//     PlcTask Inputs/GVL_iXlinker.EtherCAT_Master_EQxxxx.Beckhoff_EQ3xxx.Beckhoff_EQ3xxxEK1122.A_0006_EQ3204_0002_0016.RTD_RTDInputs_Channel_4.Status/Limit_2 <-> RTD RTDInputs Channel 4/Status/Limit 2
//     PlcTask Inputs/GVL_iXlinker.EtherCAT_Master_EQxxxx.Beckhoff_EQ3xxx.Beckhoff_EQ3xxxEK1122.A_0006_EQ3204_0002_0016.RTD_RTDInputs_Channel_1.Status/Error <-> RTD RTDInputs Channel 1/Status/Error
//     PlcTask Inputs/GVL_iXlinker.EtherCAT_Master_EQxxxx.Beckhoff_EQ3xxx.Beckhoff_EQ3xxxEK1122.A_0006_EQ3204_0002_0016.RTD_RTDInputs_Channel_2.Status/Error <-> RTD RTDInputs Channel 2/Status/Error
//     PlcTask Inputs/GVL_iXlinker.EtherCAT_Master_EQxxxx.Beckhoff_EQ3xxx.Beckhoff_EQ3xxxEK1122.A_0006_EQ3204_0002_0016.RTD_RTDInputs_Channel_3.Status/Error <-> RTD RTDInputs Channel 3/Status/Error
//     PlcTask Inputs/GVL_iXlinker.EtherCAT_Master_EQxxxx.Beckhoff_EQ3xxx.Beckhoff_EQ3xxxEK1122.A_0006_EQ3204_0002_0016.RTD_RTDInputs_Channel_4.Status/Error <-> RTD RTDInputs Channel 4/Status/Error
//     PlcTask Inputs/GVL_iXlinker.EtherCAT_Master_EQxxxx.Beckhoff_EQ3xxx.Beckhoff_EQ3xxxEK1122.A_0006_EQ3204_0002_0016.RTD_RTDInputs_Channel_1.Status/Sync_error <-> RTD RTDInputs Channel 1/Status/Sync error
//     PlcTask Inputs/GVL_iXlinker.EtherCAT_Master_EQxxxx.Beckhoff_EQ3xxx.Beckhoff_EQ3xxxEK1122.A_0006_EQ3204_0002_0016.RTD_RTDInputs_Channel_2.Status/Sync_error <-> RTD RTDInputs Channel 2/Status/Sync error
//     PlcTask Inputs/GVL_iXlinker.EtherCAT_Master_EQxxxx.Beckhoff_EQ3xxx.Beckhoff_EQ3xxxEK1122.A_0006_EQ3204_0002_0016.RTD_RTDInputs_Channel_3.Status/Sync_error <-> RTD RTDInputs Channel 3/Status/Sync error
//     PlcTask Inputs/GVL_iXlinker.EtherCAT_Master_EQxxxx.Beckhoff_EQ3xxx.Beckhoff_EQ3xxxEK1122.A_0006_EQ3204_0002_0016.RTD_RTDInputs_Channel_4.Status/Sync_error <-> RTD RTDInputs Channel 4/Status/Sync error
//     PlcTask Inputs/GVL_iXlinker.EtherCAT_Master_EQxxxx.Beckhoff_EQ3xxx.Beckhoff_EQ3xxxEK1122.A_0006_EQ3204_0002_0016.RTD_RTDInputs_Channel_1.Status/TxPDO_State <-> RTD RTDInputs Channel 1/Status/TxPDO State
//     PlcTask Inputs/GVL_iXlinker.EtherCAT_Master_EQxxxx.Beckhoff_EQ3xxx.Beckhoff_EQ3xxxEK1122.A_0006_EQ3204_0002_0016.RTD_RTDInputs_Channel_2.Status/TxPDO_State <-> RTD RTDInputs Channel 2/Status/TxPDO State
//     PlcTask Inputs/GVL_iXlinker.EtherCAT_Master_EQxxxx.Beckhoff_EQ3xxx.Beckhoff_EQ3xxxEK1122.A_0006_EQ3204_0002_0016.RTD_RTDInputs_Channel_3.Status/TxPDO_State <-> RTD RTDInputs Channel 3/Status/TxPDO State
//     PlcTask Inputs/GVL_iXlinker.EtherCAT_Master_EQxxxx.Beckhoff_EQ3xxx.Beckhoff_EQ3xxxEK1122.A_0006_EQ3204_0002_0016.RTD_RTDInputs_Channel_4.Status/TxPDO_State <-> RTD RTDInputs Channel 4/Status/TxPDO State
//     PlcTask Inputs/GVL_iXlinker.EtherCAT_Master_EQxxxx.Beckhoff_EQ3xxx.Beckhoff_EQ3xxxEK1122.A_0006_EQ3204_0002_0016.RTD_RTDInputs_Channel_1.Status/TxPDO_Toggle <-> RTD RTDInputs Channel 1/Status/TxPDO Toggle
//     PlcTask Inputs/GVL_iXlinker.EtherCAT_Master_EQxxxx.Beckhoff_EQ3xxx.Beckhoff_EQ3xxxEK1122.A_0006_EQ3204_0002_0016.RTD_RTDInputs_Channel_2.Status/TxPDO_Toggle <-> RTD RTDInputs Channel 2/Status/TxPDO Toggle
//     PlcTask Inputs/GVL_iXlinker.EtherCAT_Master_EQxxxx.Beckhoff_EQ3xxx.Beckhoff_EQ3xxxEK1122.A_0006_EQ3204_0002_0016.RTD_RTDInputs_Channel_3.Status/TxPDO_Toggle <-> RTD RTDInputs Channel 3/Status/TxPDO Toggle
//     PlcTask Inputs/GVL_iXlinker.EtherCAT_Master_EQxxxx.Beckhoff_EQ3xxx.Beckhoff_EQ3xxxEK1122.A_0006_EQ3204_0002_0016.RTD_RTDInputs_Channel_4.Status/TxPDO_Toggle <-> RTD RTDInputs Channel 4/Status/TxPDO Toggle
//     PlcTask Inputs/GVL_iXlinker.EtherCAT_Master_EQxxxx.Beckhoff_EQ3xxx.Beckhoff_EQ3xxxEK1122.A_0006_EQ3204_0002_0016.RTD_RTDInputs_Channel_1.Value <-> RTD RTDInputs Channel 1/Value
//     PlcTask Inputs/GVL_iXlinker.EtherCAT_Master_EQxxxx.Beckhoff_EQ3xxx.Beckhoff_EQ3xxxEK1122.A_0006_EQ3204_0002_0016.RTD_RTDInputs_Channel_2.Value <-> RTD RTDInputs Channel 2/Value
//     PlcTask Inputs/GVL_iXlinker.EtherCAT_Master_EQxxxx.Beckhoff_EQ3xxx.Beckhoff_EQ3xxxEK1122.A_0006_EQ3204_0002_0016.RTD_RTDInputs_Channel_3.Value <-> RTD RTDInputs Channel 3/Value
//     PlcTask Inputs/GVL_iXlinker.EtherCAT_Master_EQxxxx.Beckhoff_EQ3xxx.Beckhoff_EQ3xxxEK1122.A_0006_EQ3204_0002_0016.RTD_RTDInputs_Channel_4.Value <-> RTD RTDInputs Channel 4/Value
//     PlcTask Inputs/GVL_iXlinker.EtherCAT_Master_EQxxxx.Beckhoff_EQ3xxx.Beckhoff_EQ3xxxEK1122.A_0006_EQ3204_0002_0016.WcState.WcState <-> WcState/WcState
//     PlcTask Inputs/GVL_iXlinker.EtherCAT_Master_EQxxxx.Beckhoff_EQ3xxx.Beckhoff_EQ3xxxEK1122.A_0006_EQ3204_0002_0016.WcState.InputToggle <-> WcState/InputToggle
//     PlcTask Inputs/GVL_iXlinker.EtherCAT_Master_EQxxxx.Beckhoff_EQ3xxx.Beckhoff_EQ3xxxEK1122.A_0006_EQ3204_0002_0016.InfoData.AdsAddr <-> InfoData/AdsAddr
//     PlcTask Inputs/GVL_iXlinker.EtherCAT_Master_EQxxxx.Beckhoff_EQ3xxx.Beckhoff_EQ3xxxEK1122.A_0006_EQ3204_0002_0016.InfoData.State <-> InfoData/State
//   PLC/PLC Instance <-> EtherCAT Master EQxxxx/Beckhoff EQ3xxx/Beckhoff EQ3xxxEK1122/A_0007(EQ3204-0002-0017)
//     PlcTask Inputs/GVL_iXlinker.EtherCAT_Master_EQxxxx.Beckhoff_EQ3xxx.Beckhoff_EQ3xxxEK1122.A_0007_EQ3204_0002_0017.RTD_RTDInputs_Channel_1.Status/Underrange <-> RTD RTDInputs Channel 1/Status/Underrange
//     PlcTask Inputs/GVL_iXlinker.EtherCAT_Master_EQxxxx.Beckhoff_EQ3xxx.Beckhoff_EQ3xxxEK1122.A_0007_EQ3204_0002_0017.RTD_RTDInputs_Channel_2.Status/Underrange <-> RTD RTDInputs Channel 2/Status/Underrange
//     PlcTask Inputs/GVL_iXlinker.EtherCAT_Master_EQxxxx.Beckhoff_EQ3xxx.Beckhoff_EQ3xxxEK1122.A_0007_EQ3204_0002_0017.RTD_RTDInputs_Channel_3.Status/Underrange <-> RTD RTDInputs Channel 3/Status/Underrange
//     PlcTask Inputs/GVL_iXlinker.EtherCAT_Master_EQxxxx.Beckhoff_EQ3xxx.Beckhoff_EQ3xxxEK1122.A_0007_EQ3204_0002_0017.RTD_RTDInputs_Channel_4.Status/Underrange <-> RTD RTDInputs Channel 4/Status/Underrange
//     PlcTask Inputs/GVL_iXlinker.EtherCAT_Master_EQxxxx.Beckhoff_EQ3xxx.Beckhoff_EQ3xxxEK1122.A_0007_EQ3204_0002_0017.RTD_RTDInputs_Channel_1.Status/Overrange <-> RTD RTDInputs Channel 1/Status/Overrange
//     PlcTask Inputs/GVL_iXlinker.EtherCAT_Master_EQxxxx.Beckhoff_EQ3xxx.Beckhoff_EQ3xxxEK1122.A_0007_EQ3204_0002_0017.RTD_RTDInputs_Channel_2.Status/Overrange <-> RTD RTDInputs Channel 2/Status/Overrange
//     PlcTask Inputs/GVL_iXlinker.EtherCAT_Master_EQxxxx.Beckhoff_EQ3xxx.Beckhoff_EQ3xxxEK1122.A_0007_EQ3204_0002_0017.RTD_RTDInputs_Channel_3.Status/Overrange <-> RTD RTDInputs Channel 3/Status/Overrange
//     PlcTask Inputs/GVL_iXlinker.EtherCAT_Master_EQxxxx.Beckhoff_EQ3xxx.Beckhoff_EQ3xxxEK1122.A_0007_EQ3204_0002_0017.RTD_RTDInputs_Channel_4.Status/Overrange <-> RTD RTDInputs Channel 4/Status/Overrange
//     PlcTask Inputs/GVL_iXlinker.EtherCAT_Master_EQxxxx.Beckhoff_EQ3xxx.Beckhoff_EQ3xxxEK1122.A_0007_EQ3204_0002_0017.RTD_RTDInputs_Channel_1.Status/Limit_1 <-> RTD RTDInputs Channel 1/Status/Limit 1
//     PlcTask Inputs/GVL_iXlinker.EtherCAT_Master_EQxxxx.Beckhoff_EQ3xxx.Beckhoff_EQ3xxxEK1122.A_0007_EQ3204_0002_0017.RTD_RTDInputs_Channel_1.Status/Limit_2 <-> RTD RTDInputs Channel 1/Status/Limit 2
//     PlcTask Inputs/GVL_iXlinker.EtherCAT_Master_EQxxxx.Beckhoff_EQ3xxx.Beckhoff_EQ3xxxEK1122.A_0007_EQ3204_0002_0017.RTD_RTDInputs_Channel_2.Status/Limit_1 <-> RTD RTDInputs Channel 2/Status/Limit 1
//     PlcTask Inputs/GVL_iXlinker.EtherCAT_Master_EQxxxx.Beckhoff_EQ3xxx.Beckhoff_EQ3xxxEK1122.A_0007_EQ3204_0002_0017.RTD_RTDInputs_Channel_2.Status/Limit_2 <-> RTD RTDInputs Channel 2/Status/Limit 2
//     PlcTask Inputs/GVL_iXlinker.EtherCAT_Master_EQxxxx.Beckhoff_EQ3xxx.Beckhoff_EQ3xxxEK1122.A_0007_EQ3204_0002_0017.RTD_RTDInputs_Channel_3.Status/Limit_1 <-> RTD RTDInputs Channel 3/Status/Limit 1
//     PlcTask Inputs/GVL_iXlinker.EtherCAT_Master_EQxxxx.Beckhoff_EQ3xxx.Beckhoff_EQ3xxxEK1122.A_0007_EQ3204_0002_0017.RTD_RTDInputs_Channel_3.Status/Limit_2 <-> RTD RTDInputs Channel 3/Status/Limit 2
//     PlcTask Inputs/GVL_iXlinker.EtherCAT_Master_EQxxxx.Beckhoff_EQ3xxx.Beckhoff_EQ3xxxEK1122.A_0007_EQ3204_0002_0017.RTD_RTDInputs_Channel_4.Status/Limit_1 <-> RTD RTDInputs Channel 4/Status/Limit 1
//     PlcTask Inputs/GVL_iXlinker.EtherCAT_Master_EQxxxx.Beckhoff_EQ3xxx.Beckhoff_EQ3xxxEK1122.A_0007_EQ3204_0002_0017.RTD_RTDInputs_Channel_4.Status/Limit_2 <-> RTD RTDInputs Channel 4/Status/Limit 2
//     PlcTask Inputs/GVL_iXlinker.EtherCAT_Master_EQxxxx.Beckhoff_EQ3xxx.Beckhoff_EQ3xxxEK1122.A_0007_EQ3204_0002_0017.RTD_RTDInputs_Channel_1.Status/Error <-> RTD RTDInputs Channel 1/Status/Error
//     PlcTask Inputs/GVL_iXlinker.EtherCAT_Master_EQxxxx.Beckhoff_EQ3xxx.Beckhoff_EQ3xxxEK1122.A_0007_EQ3204_0002_0017.RTD_RTDInputs_Channel_2.Status/Error <-> RTD RTDInputs Channel 2/Status/Error
//     PlcTask Inputs/GVL_iXlinker.EtherCAT_Master_EQxxxx.Beckhoff_EQ3xxx.Beckhoff_EQ3xxxEK1122.A_0007_EQ3204_0002_0017.RTD_RTDInputs_Channel_3.Status/Error <-> RTD RTDInputs Channel 3/Status/Error
//     PlcTask Inputs/GVL_iXlinker.EtherCAT_Master_EQxxxx.Beckhoff_EQ3xxx.Beckhoff_EQ3xxxEK1122.A_0007_EQ3204_0002_0017.RTD_RTDInputs_Channel_4.Status/Error <-> RTD RTDInputs Channel 4/Status/Error
//     PlcTask Inputs/GVL_iXlinker.EtherCAT_Master_EQxxxx.Beckhoff_EQ3xxx.Beckhoff_EQ3xxxEK1122.A_0007_EQ3204_0002_0017.RTD_RTDInputs_Channel_1.Status/Sync_error <-> RTD RTDInputs Channel 1/Status/Sync error
//     PlcTask Inputs/GVL_iXlinker.EtherCAT_Master_EQxxxx.Beckhoff_EQ3xxx.Beckhoff_EQ3xxxEK1122.A_0007_EQ3204_0002_0017.RTD_RTDInputs_Channel_2.Status/Sync_error <-> RTD RTDInputs Channel 2/Status/Sync error
//     PlcTask Inputs/GVL_iXlinker.EtherCAT_Master_EQxxxx.Beckhoff_EQ3xxx.Beckhoff_EQ3xxxEK1122.A_0007_EQ3204_0002_0017.RTD_RTDInputs_Channel_3.Status/Sync_error <-> RTD RTDInputs Channel 3/Status/Sync error
//     PlcTask Inputs/GVL_iXlinker.EtherCAT_Master_EQxxxx.Beckhoff_EQ3xxx.Beckhoff_EQ3xxxEK1122.A_0007_EQ3204_0002_0017.RTD_RTDInputs_Channel_4.Status/Sync_error <-> RTD RTDInputs Channel 4/Status/Sync error
//     PlcTask Inputs/GVL_iXlinker.EtherCAT_Master_EQxxxx.Beckhoff_EQ3xxx.Beckhoff_EQ3xxxEK1122.A_0007_EQ3204_0002_0017.RTD_RTDInputs_Channel_1.Status/TxPDO_State <-> RTD RTDInputs Channel 1/Status/TxPDO State
//     PlcTask Inputs/GVL_iXlinker.EtherCAT_Master_EQxxxx.Beckhoff_EQ3xxx.Beckhoff_EQ3xxxEK1122.A_0007_EQ3204_0002_0017.RTD_RTDInputs_Channel_2.Status/TxPDO_State <-> RTD RTDInputs Channel 2/Status/TxPDO State
//     PlcTask Inputs/GVL_iXlinker.EtherCAT_Master_EQxxxx.Beckhoff_EQ3xxx.Beckhoff_EQ3xxxEK1122.A_0007_EQ3204_0002_0017.RTD_RTDInputs_Channel_3.Status/TxPDO_State <-> RTD RTDInputs Channel 3/Status/TxPDO State
//     PlcTask Inputs/GVL_iXlinker.EtherCAT_Master_EQxxxx.Beckhoff_EQ3xxx.Beckhoff_EQ3xxxEK1122.A_0007_EQ3204_0002_0017.RTD_RTDInputs_Channel_4.Status/TxPDO_State <-> RTD RTDInputs Channel 4/Status/TxPDO State
//     PlcTask Inputs/GVL_iXlinker.EtherCAT_Master_EQxxxx.Beckhoff_EQ3xxx.Beckhoff_EQ3xxxEK1122.A_0007_EQ3204_0002_0017.RTD_RTDInputs_Channel_1.Status/TxPDO_Toggle <-> RTD RTDInputs Channel 1/Status/TxPDO Toggle
//     PlcTask Inputs/GVL_iXlinker.EtherCAT_Master_EQxxxx.Beckhoff_EQ3xxx.Beckhoff_EQ3xxxEK1122.A_0007_EQ3204_0002_0017.RTD_RTDInputs_Channel_2.Status/TxPDO_Toggle <-> RTD RTDInputs Channel 2/Status/TxPDO Toggle
//     PlcTask Inputs/GVL_iXlinker.EtherCAT_Master_EQxxxx.Beckhoff_EQ3xxx.Beckhoff_EQ3xxxEK1122.A_0007_EQ3204_0002_0017.RTD_RTDInputs_Channel_3.Status/TxPDO_Toggle <-> RTD RTDInputs Channel 3/Status/TxPDO Toggle
//     PlcTask Inputs/GVL_iXlinker.EtherCAT_Master_EQxxxx.Beckhoff_EQ3xxx.Beckhoff_EQ3xxxEK1122.A_0007_EQ3204_0002_0017.RTD_RTDInputs_Channel_4.Status/TxPDO_Toggle <-> RTD RTDInputs Channel 4/Status/TxPDO Toggle
//     PlcTask Inputs/GVL_iXlinker.EtherCAT_Master_EQxxxx.Beckhoff_EQ3xxx.Beckhoff_EQ3xxxEK1122.A_0007_EQ3204_0002_0017.RTD_RTDInputs_Channel_1.Value <-> RTD RTDInputs Channel 1/Value
//     PlcTask Inputs/GVL_iXlinker.EtherCAT_Master_EQxxxx.Beckhoff_EQ3xxx.Beckhoff_EQ3xxxEK1122.A_0007_EQ3204_0002_0017.RTD_RTDInputs_Channel_2.Value <-> RTD RTDInputs Channel 2/Value
//     PlcTask Inputs/GVL_iXlinker.EtherCAT_Master_EQxxxx.Beckhoff_EQ3xxx.Beckhoff_EQ3xxxEK1122.A_0007_EQ3204_0002_0017.RTD_RTDInputs_Channel_3.Value <-> RTD RTDInputs Channel 3/Value
//     PlcTask Inputs/GVL_iXlinker.EtherCAT_Master_EQxxxx.Beckhoff_EQ3xxx.Beckhoff_EQ3xxxEK1122.A_0007_EQ3204_0002_0017.RTD_RTDInputs_Channel_4.Value <-> RTD RTDInputs Channel 4/Value
//     PlcTask Inputs/GVL_iXlinker.EtherCAT_Master_EQxxxx.Beckhoff_EQ3xxx.Beckhoff_EQ3xxxEK1122.A_0007_EQ3204_0002_0017.WcState.WcState <-> WcState/WcState
//     PlcTask Inputs/GVL_iXlinker.EtherCAT_Master_EQxxxx.Beckhoff_EQ3xxx.Beckhoff_EQ3xxxEK1122.A_0007_EQ3204_0002_0017.WcState.InputToggle <-> WcState/InputToggle
//     PlcTask Inputs/GVL_iXlinker.EtherCAT_Master_EQxxxx.Beckhoff_EQ3xxx.Beckhoff_EQ3xxxEK1122.A_0007_EQ3204_0002_0017.InfoData.AdsAddr <-> InfoData/AdsAddr
//     PlcTask Inputs/GVL_iXlinker.EtherCAT_Master_EQxxxx.Beckhoff_EQ3xxx.Beckhoff_EQ3xxxEK1122.A_0007_EQ3204_0002_0017.InfoData.State <-> InfoData/State
//   PLC/PLC Instance <-> EtherCAT Master EQxxxx/Beckhoff EQ3xxx/Beckhoff EQ3xxxEK1122/A_0008(EQ3204-0002-0020)
//     PlcTask Inputs/GVL_iXlinker.EtherCAT_Master_EQxxxx.Beckhoff_EQ3xxx.Beckhoff_EQ3xxxEK1122.A_0008_EQ3204_0002_0020.RTD_RTDInputs_Channel_1.Status/Underrange <-> RTD RTDInputs Channel 1/Status/Underrange
//     PlcTask Inputs/GVL_iXlinker.EtherCAT_Master_EQxxxx.Beckhoff_EQ3xxx.Beckhoff_EQ3xxxEK1122.A_0008_EQ3204_0002_0020.RTD_RTDInputs_Channel_2.Status/Underrange <-> RTD RTDInputs Channel 2/Status/Underrange
//     PlcTask Inputs/GVL_iXlinker.EtherCAT_Master_EQxxxx.Beckhoff_EQ3xxx.Beckhoff_EQ3xxxEK1122.A_0008_EQ3204_0002_0020.RTD_RTDInputs_Channel_3.Status/Underrange <-> RTD RTDInputs Channel 3/Status/Underrange
//     PlcTask Inputs/GVL_iXlinker.EtherCAT_Master_EQxxxx.Beckhoff_EQ3xxx.Beckhoff_EQ3xxxEK1122.A_0008_EQ3204_0002_0020.RTD_RTDInputs_Channel_4.Status/Underrange <-> RTD RTDInputs Channel 4/Status/Underrange
//     PlcTask Inputs/GVL_iXlinker.EtherCAT_Master_EQxxxx.Beckhoff_EQ3xxx.Beckhoff_EQ3xxxEK1122.A_0008_EQ3204_0002_0020.RTD_RTDInputs_Channel_1.Status/Overrange <-> RTD RTDInputs Channel 1/Status/Overrange
//     PlcTask Inputs/GVL_iXlinker.EtherCAT_Master_EQxxxx.Beckhoff_EQ3xxx.Beckhoff_EQ3xxxEK1122.A_0008_EQ3204_0002_0020.RTD_RTDInputs_Channel_2.Status/Overrange <-> RTD RTDInputs Channel 2/Status/Overrange
//     PlcTask Inputs/GVL_iXlinker.EtherCAT_Master_EQxxxx.Beckhoff_EQ3xxx.Beckhoff_EQ3xxxEK1122.A_0008_EQ3204_0002_0020.RTD_RTDInputs_Channel_3.Status/Overrange <-> RTD RTDInputs Channel 3/Status/Overrange
//     PlcTask Inputs/GVL_iXlinker.EtherCAT_Master_EQxxxx.Beckhoff_EQ3xxx.Beckhoff_EQ3xxxEK1122.A_0008_EQ3204_0002_0020.RTD_RTDInputs_Channel_4.Status/Overrange <-> RTD RTDInputs Channel 4/Status/Overrange
//     PlcTask Inputs/GVL_iXlinker.EtherCAT_Master_EQxxxx.Beckhoff_EQ3xxx.Beckhoff_EQ3xxxEK1122.A_0008_EQ3204_0002_0020.RTD_RTDInputs_Channel_1.Status/Limit_1 <-> RTD RTDInputs Channel 1/Status/Limit 1
//     PlcTask Inputs/GVL_iXlinker.EtherCAT_Master_EQxxxx.Beckhoff_EQ3xxx.Beckhoff_EQ3xxxEK1122.A_0008_EQ3204_0002_0020.RTD_RTDInputs_Channel_1.Status/Limit_2 <-> RTD RTDInputs Channel 1/Status/Limit 2
//     PlcTask Inputs/GVL_iXlinker.EtherCAT_Master_EQxxxx.Beckhoff_EQ3xxx.Beckhoff_EQ3xxxEK1122.A_0008_EQ3204_0002_0020.RTD_RTDInputs_Channel_2.Status/Limit_1 <-> RTD RTDInputs Channel 2/Status/Limit 1
//     PlcTask Inputs/GVL_iXlinker.EtherCAT_Master_EQxxxx.Beckhoff_EQ3xxx.Beckhoff_EQ3xxxEK1122.A_0008_EQ3204_0002_0020.RTD_RTDInputs_Channel_2.Status/Limit_2 <-> RTD RTDInputs Channel 2/Status/Limit 2
//     PlcTask Inputs/GVL_iXlinker.EtherCAT_Master_EQxxxx.Beckhoff_EQ3xxx.Beckhoff_EQ3xxxEK1122.A_0008_EQ3204_0002_0020.RTD_RTDInputs_Channel_3.Status/Limit_1 <-> RTD RTDInputs Channel 3/Status/Limit 1
//     PlcTask Inputs/GVL_iXlinker.EtherCAT_Master_EQxxxx.Beckhoff_EQ3xxx.Beckhoff_EQ3xxxEK1122.A_0008_EQ3204_0002_0020.RTD_RTDInputs_Channel_3.Status/Limit_2 <-> RTD RTDInputs Channel 3/Status/Limit 2
//     PlcTask Inputs/GVL_iXlinker.EtherCAT_Master_EQxxxx.Beckhoff_EQ3xxx.Beckhoff_EQ3xxxEK1122.A_0008_EQ3204_0002_0020.RTD_RTDInputs_Channel_4.Status/Limit_1 <-> RTD RTDInputs Channel 4/Status/Limit 1
//     PlcTask Inputs/GVL_iXlinker.EtherCAT_Master_EQxxxx.Beckhoff_EQ3xxx.Beckhoff_EQ3xxxEK1122.A_0008_EQ3204_0002_0020.RTD_RTDInputs_Channel_4.Status/Limit_2 <-> RTD RTDInputs Channel 4/Status/Limit 2
//     PlcTask Inputs/GVL_iXlinker.EtherCAT_Master_EQxxxx.Beckhoff_EQ3xxx.Beckhoff_EQ3xxxEK1122.A_0008_EQ3204_0002_0020.RTD_RTDInputs_Channel_1.Status/Error <-> RTD RTDInputs Channel 1/Status/Error
//     PlcTask Inputs/GVL_iXlinker.EtherCAT_Master_EQxxxx.Beckhoff_EQ3xxx.Beckhoff_EQ3xxxEK1122.A_0008_EQ3204_0002_0020.RTD_RTDInputs_Channel_2.Status/Error <-> RTD RTDInputs Channel 2/Status/Error
//     PlcTask Inputs/GVL_iXlinker.EtherCAT_Master_EQxxxx.Beckhoff_EQ3xxx.Beckhoff_EQ3xxxEK1122.A_0008_EQ3204_0002_0020.RTD_RTDInputs_Channel_3.Status/Error <-> RTD RTDInputs Channel 3/Status/Error
//     PlcTask Inputs/GVL_iXlinker.EtherCAT_Master_EQxxxx.Beckhoff_EQ3xxx.Beckhoff_EQ3xxxEK1122.A_0008_EQ3204_0002_0020.RTD_RTDInputs_Channel_4.Status/Error <-> RTD RTDInputs Channel 4/Status/Error
//     PlcTask Inputs/GVL_iXlinker.EtherCAT_Master_EQxxxx.Beckhoff_EQ3xxx.Beckhoff_EQ3xxxEK1122.A_0008_EQ3204_0002_0020.RTD_RTDInputs_Channel_1.Status/Sync_error <-> RTD RTDInputs Channel 1/Status/Sync error
//     PlcTask Inputs/GVL_iXlinker.EtherCAT_Master_EQxxxx.Beckhoff_EQ3xxx.Beckhoff_EQ3xxxEK1122.A_0008_EQ3204_0002_0020.RTD_RTDInputs_Channel_2.Status/Sync_error <-> RTD RTDInputs Channel 2/Status/Sync error
//     PlcTask Inputs/GVL_iXlinker.EtherCAT_Master_EQxxxx.Beckhoff_EQ3xxx.Beckhoff_EQ3xxxEK1122.A_0008_EQ3204_0002_0020.RTD_RTDInputs_Channel_3.Status/Sync_error <-> RTD RTDInputs Channel 3/Status/Sync error
//     PlcTask Inputs/GVL_iXlinker.EtherCAT_Master_EQxxxx.Beckhoff_EQ3xxx.Beckhoff_EQ3xxxEK1122.A_0008_EQ3204_0002_0020.RTD_RTDInputs_Channel_4.Status/Sync_error <-> RTD RTDInputs Channel 4/Status/Sync error
//     PlcTask Inputs/GVL_iXlinker.EtherCAT_Master_EQxxxx.Beckhoff_EQ3xxx.Beckhoff_EQ3xxxEK1122.A_0008_EQ3204_0002_0020.RTD_RTDInputs_Channel_1.Status/TxPDO_State <-> RTD RTDInputs Channel 1/Status/TxPDO State
//     PlcTask Inputs/GVL_iXlinker.EtherCAT_Master_EQxxxx.Beckhoff_EQ3xxx.Beckhoff_EQ3xxxEK1122.A_0008_EQ3204_0002_0020.RTD_RTDInputs_Channel_2.Status/TxPDO_State <-> RTD RTDInputs Channel 2/Status/TxPDO State
//     PlcTask Inputs/GVL_iXlinker.EtherCAT_Master_EQxxxx.Beckhoff_EQ3xxx.Beckhoff_EQ3xxxEK1122.A_0008_EQ3204_0002_0020.RTD_RTDInputs_Channel_3.Status/TxPDO_State <-> RTD RTDInputs Channel 3/Status/TxPDO State
//     PlcTask Inputs/GVL_iXlinker.EtherCAT_Master_EQxxxx.Beckhoff_EQ3xxx.Beckhoff_EQ3xxxEK1122.A_0008_EQ3204_0002_0020.RTD_RTDInputs_Channel_4.Status/TxPDO_State <-> RTD RTDInputs Channel 4/Status/TxPDO State
//     PlcTask Inputs/GVL_iXlinker.EtherCAT_Master_EQxxxx.Beckhoff_EQ3xxx.Beckhoff_EQ3xxxEK1122.A_0008_EQ3204_0002_0020.RTD_RTDInputs_Channel_1.Status/TxPDO_Toggle <-> RTD RTDInputs Channel 1/Status/TxPDO Toggle
//     PlcTask Inputs/GVL_iXlinker.EtherCAT_Master_EQxxxx.Beckhoff_EQ3xxx.Beckhoff_EQ3xxxEK1122.A_0008_EQ3204_0002_0020.RTD_RTDInputs_Channel_2.Status/TxPDO_Toggle <-> RTD RTDInputs Channel 2/Status/TxPDO Toggle
//     PlcTask Inputs/GVL_iXlinker.EtherCAT_Master_EQxxxx.Beckhoff_EQ3xxx.Beckhoff_EQ3xxxEK1122.A_0008_EQ3204_0002_0020.RTD_RTDInputs_Channel_3.Status/TxPDO_Toggle <-> RTD RTDInputs Channel 3/Status/TxPDO Toggle
//     PlcTask Inputs/GVL_iXlinker.EtherCAT_Master_EQxxxx.Beckhoff_EQ3xxx.Beckhoff_EQ3xxxEK1122.A_0008_EQ3204_0002_0020.RTD_RTDInputs_Channel_4.Status/TxPDO_Toggle <-> RTD RTDInputs Channel 4/Status/TxPDO Toggle
//     PlcTask Inputs/GVL_iXlinker.EtherCAT_Master_EQxxxx.Beckhoff_EQ3xxx.Beckhoff_EQ3xxxEK1122.A_0008_EQ3204_0002_0020.RTD_RTDInputs_Channel_1.Value <-> RTD RTDInputs Channel 1/Value
//     PlcTask Inputs/GVL_iXlinker.EtherCAT_Master_EQxxxx.Beckhoff_EQ3xxx.Beckhoff_EQ3xxxEK1122.A_0008_EQ3204_0002_0020.RTD_RTDInputs_Channel_2.Value <-> RTD RTDInputs Channel 2/Value
//     PlcTask Inputs/GVL_iXlinker.EtherCAT_Master_EQxxxx.Beckhoff_EQ3xxx.Beckhoff_EQ3xxxEK1122.A_0008_EQ3204_0002_0020.RTD_RTDInputs_Channel_3.Value <-> RTD RTDInputs Channel 3/Value
//     PlcTask Inputs/GVL_iXlinker.EtherCAT_Master_EQxxxx.Beckhoff_EQ3xxx.Beckhoff_EQ3xxxEK1122.A_0008_EQ3204_0002_0020.RTD_RTDInputs_Channel_4.Value <-> RTD RTDInputs Channel 4/Value
//     PlcTask Inputs/GVL_iXlinker.EtherCAT_Master_EQxxxx.Beckhoff_EQ3xxx.Beckhoff_EQ3xxxEK1122.A_0008_EQ3204_0002_0020.WcState.WcState <-> WcState/WcState
//     PlcTask Inputs/GVL_iXlinker.EtherCAT_Master_EQxxxx.Beckhoff_EQ3xxx.Beckhoff_EQ3xxxEK1122.A_0008_EQ3204_0002_0020.WcState.InputToggle <-> WcState/InputToggle
//     PlcTask Inputs/GVL_iXlinker.EtherCAT_Master_EQxxxx.Beckhoff_EQ3xxx.Beckhoff_EQ3xxxEK1122.A_0008_EQ3204_0002_0020.InfoData.AdsAddr <-> InfoData/AdsAddr
//     PlcTask Inputs/GVL_iXlinker.EtherCAT_Master_EQxxxx.Beckhoff_EQ3xxx.Beckhoff_EQ3xxxEK1122.A_0008_EQ3204_0002_0020.InfoData.State <-> InfoData/State
//   PLC/PLC Instance <-> EtherCAT Master EQxxxx/Beckhoff EQ3xxx/Beckhoff EQ3xxxEK1122/A_0009(EQ3204-0002-0021)
//     PlcTask Inputs/GVL_iXlinker.EtherCAT_Master_EQxxxx.Beckhoff_EQ3xxx.Beckhoff_EQ3xxxEK1122.A_0009_EQ3204_0002_0021.RTD_RTDInputs_Channel_1.Status/Underrange <-> RTD RTDInputs Channel 1/Status/Underrange
//     PlcTask Inputs/GVL_iXlinker.EtherCAT_Master_EQxxxx.Beckhoff_EQ3xxx.Beckhoff_EQ3xxxEK1122.A_0009_EQ3204_0002_0021.RTD_RTDInputs_Channel_2.Status/Underrange <-> RTD RTDInputs Channel 2/Status/Underrange
//     PlcTask Inputs/GVL_iXlinker.EtherCAT_Master_EQxxxx.Beckhoff_EQ3xxx.Beckhoff_EQ3xxxEK1122.A_0009_EQ3204_0002_0021.RTD_RTDInputs_Channel_3.Status/Underrange <-> RTD RTDInputs Channel 3/Status/Underrange
//     PlcTask Inputs/GVL_iXlinker.EtherCAT_Master_EQxxxx.Beckhoff_EQ3xxx.Beckhoff_EQ3xxxEK1122.A_0009_EQ3204_0002_0021.RTD_RTDInputs_Channel_4.Status/Underrange <-> RTD RTDInputs Channel 4/Status/Underrange
//     PlcTask Inputs/GVL_iXlinker.EtherCAT_Master_EQxxxx.Beckhoff_EQ3xxx.Beckhoff_EQ3xxxEK1122.A_0009_EQ3204_0002_0021.RTD_RTDInputs_Channel_1.Status/Overrange <-> RTD RTDInputs Channel 1/Status/Overrange
//     PlcTask Inputs/GVL_iXlinker.EtherCAT_Master_EQxxxx.Beckhoff_EQ3xxx.Beckhoff_EQ3xxxEK1122.A_0009_EQ3204_0002_0021.RTD_RTDInputs_Channel_2.Status/Overrange <-> RTD RTDInputs Channel 2/Status/Overrange
//     PlcTask Inputs/GVL_iXlinker.EtherCAT_Master_EQxxxx.Beckhoff_EQ3xxx.Beckhoff_EQ3xxxEK1122.A_0009_EQ3204_0002_0021.RTD_RTDInputs_Channel_3.Status/Overrange <-> RTD RTDInputs Channel 3/Status/Overrange
//     PlcTask Inputs/GVL_iXlinker.EtherCAT_Master_EQxxxx.Beckhoff_EQ3xxx.Beckhoff_EQ3xxxEK1122.A_0009_EQ3204_0002_0021.RTD_RTDInputs_Channel_4.Status/Overrange <-> RTD RTDInputs Channel 4/Status/Overrange
//     PlcTask Inputs/GVL_iXlinker.EtherCAT_Master_EQxxxx.Beckhoff_EQ3xxx.Beckhoff_EQ3xxxEK1122.A_0009_EQ3204_0002_0021.RTD_RTDInputs_Channel_1.Status/Limit_1 <-> RTD RTDInputs Channel 1/Status/Limit 1
//     PlcTask Inputs/GVL_iXlinker.EtherCAT_Master_EQxxxx.Beckhoff_EQ3xxx.Beckhoff_EQ3xxxEK1122.A_0009_EQ3204_0002_0021.RTD_RTDInputs_Channel_1.Status/Limit_2 <-> RTD RTDInputs Channel 1/Status/Limit 2
//     PlcTask Inputs/GVL_iXlinker.EtherCAT_Master_EQxxxx.Beckhoff_EQ3xxx.Beckhoff_EQ3xxxEK1122.A_0009_EQ3204_0002_0021.RTD_RTDInputs_Channel_2.Status/Limit_1 <-> RTD RTDInputs Channel 2/Status/Limit 1
//     PlcTask Inputs/GVL_iXlinker.EtherCAT_Master_EQxxxx.Beckhoff_EQ3xxx.Beckhoff_EQ3xxxEK1122.A_0009_EQ3204_0002_0021.RTD_RTDInputs_Channel_2.Status/Limit_2 <-> RTD RTDInputs Channel 2/Status/Limit 2
//     PlcTask Inputs/GVL_iXlinker.EtherCAT_Master_EQxxxx.Beckhoff_EQ3xxx.Beckhoff_EQ3xxxEK1122.A_0009_EQ3204_0002_0021.RTD_RTDInputs_Channel_3.Status/Limit_1 <-> RTD RTDInputs Channel 3/Status/Limit 1
//     PlcTask Inputs/GVL_iXlinker.EtherCAT_Master_EQxxxx.Beckhoff_EQ3xxx.Beckhoff_EQ3xxxEK1122.A_0009_EQ3204_0002_0021.RTD_RTDInputs_Channel_3.Status/Limit_2 <-> RTD RTDInputs Channel 3/Status/Limit 2
//     PlcTask Inputs/GVL_iXlinker.EtherCAT_Master_EQxxxx.Beckhoff_EQ3xxx.Beckhoff_EQ3xxxEK1122.A_0009_EQ3204_0002_0021.RTD_RTDInputs_Channel_4.Status/Limit_1 <-> RTD RTDInputs Channel 4/Status/Limit 1
//     PlcTask Inputs/GVL_iXlinker.EtherCAT_Master_EQxxxx.Beckhoff_EQ3xxx.Beckhoff_EQ3xxxEK1122.A_0009_EQ3204_0002_0021.RTD_RTDInputs_Channel_4.Status/Limit_2 <-> RTD RTDInputs Channel 4/Status/Limit 2
//     PlcTask Inputs/GVL_iXlinker.EtherCAT_Master_EQxxxx.Beckhoff_EQ3xxx.Beckhoff_EQ3xxxEK1122.A_0009_EQ3204_0002_0021.RTD_RTDInputs_Channel_1.Status/Error <-> RTD RTDInputs Channel 1/Status/Error
//     PlcTask Inputs/GVL_iXlinker.EtherCAT_Master_EQxxxx.Beckhoff_EQ3xxx.Beckhoff_EQ3xxxEK1122.A_0009_EQ3204_0002_0021.RTD_RTDInputs_Channel_2.Status/Error <-> RTD RTDInputs Channel 2/Status/Error
//     PlcTask Inputs/GVL_iXlinker.EtherCAT_Master_EQxxxx.Beckhoff_EQ3xxx.Beckhoff_EQ3xxxEK1122.A_0009_EQ3204_0002_0021.RTD_RTDInputs_Channel_3.Status/Error <-> RTD RTDInputs Channel 3/Status/Error
//     PlcTask Inputs/GVL_iXlinker.EtherCAT_Master_EQxxxx.Beckhoff_EQ3xxx.Beckhoff_EQ3xxxEK1122.A_0009_EQ3204_0002_0021.RTD_RTDInputs_Channel_4.Status/Error <-> RTD RTDInputs Channel 4/Status/Error
//     PlcTask Inputs/GVL_iXlinker.EtherCAT_Master_EQxxxx.Beckhoff_EQ3xxx.Beckhoff_EQ3xxxEK1122.A_0009_EQ3204_0002_0021.RTD_RTDInputs_Channel_1.Status/TxPDO_State <-> RTD RTDInputs Channel 1/Status/TxPDO State
//     PlcTask Inputs/GVL_iXlinker.EtherCAT_Master_EQxxxx.Beckhoff_EQ3xxx.Beckhoff_EQ3xxxEK1122.A_0009_EQ3204_0002_0021.RTD_RTDInputs_Channel_2.Status/TxPDO_State <-> RTD RTDInputs Channel 2/Status/TxPDO State
//     PlcTask Inputs/GVL_iXlinker.EtherCAT_Master_EQxxxx.Beckhoff_EQ3xxx.Beckhoff_EQ3xxxEK1122.A_0009_EQ3204_0002_0021.RTD_RTDInputs_Channel_3.Status/TxPDO_State <-> RTD RTDInputs Channel 3/Status/TxPDO State
//     PlcTask Inputs/GVL_iXlinker.EtherCAT_Master_EQxxxx.Beckhoff_EQ3xxx.Beckhoff_EQ3xxxEK1122.A_0009_EQ3204_0002_0021.RTD_RTDInputs_Channel_4.Status/TxPDO_State <-> RTD RTDInputs Channel 4/Status/TxPDO State
//     PlcTask Inputs/GVL_iXlinker.EtherCAT_Master_EQxxxx.Beckhoff_EQ3xxx.Beckhoff_EQ3xxxEK1122.A_0009_EQ3204_0002_0021.RTD_RTDInputs_Channel_1.Status/TxPDO_Toggle <-> RTD RTDInputs Channel 1/Status/TxPDO Toggle
//     PlcTask Inputs/GVL_iXlinker.EtherCAT_Master_EQxxxx.Beckhoff_EQ3xxx.Beckhoff_EQ3xxxEK1122.A_0009_EQ3204_0002_0021.RTD_RTDInputs_Channel_2.Status/TxPDO_Toggle <-> RTD RTDInputs Channel 2/Status/TxPDO Toggle
//     PlcTask Inputs/GVL_iXlinker.EtherCAT_Master_EQxxxx.Beckhoff_EQ3xxx.Beckhoff_EQ3xxxEK1122.A_0009_EQ3204_0002_0021.RTD_RTDInputs_Channel_3.Status/TxPDO_Toggle <-> RTD RTDInputs Channel 3/Status/TxPDO Toggle
//     PlcTask Inputs/GVL_iXlinker.EtherCAT_Master_EQxxxx.Beckhoff_EQ3xxx.Beckhoff_EQ3xxxEK1122.A_0009_EQ3204_0002_0021.RTD_RTDInputs_Channel_4.Status/TxPDO_Toggle <-> RTD RTDInputs Channel 4/Status/TxPDO Toggle
//     PlcTask Inputs/GVL_iXlinker.EtherCAT_Master_EQxxxx.Beckhoff_EQ3xxx.Beckhoff_EQ3xxxEK1122.A_0009_EQ3204_0002_0021.RTD_RTDInputs_Channel_1.Value <-> RTD RTDInputs Channel 1/Value
//     PlcTask Inputs/GVL_iXlinker.EtherCAT_Master_EQxxxx.Beckhoff_EQ3xxx.Beckhoff_EQ3xxxEK1122.A_0009_EQ3204_0002_0021.RTD_RTDInputs_Channel_2.Value <-> RTD RTDInputs Channel 2/Value
//     PlcTask Inputs/GVL_iXlinker.EtherCAT_Master_EQxxxx.Beckhoff_EQ3xxx.Beckhoff_EQ3xxxEK1122.A_0009_EQ3204_0002_0021.RTD_RTDInputs_Channel_3.Value <-> RTD RTDInputs Channel 3/Value
//     PlcTask Inputs/GVL_iXlinker.EtherCAT_Master_EQxxxx.Beckhoff_EQ3xxx.Beckhoff_EQ3xxxEK1122.A_0009_EQ3204_0002_0021.RTD_RTDInputs_Channel_4.Value <-> RTD RTDInputs Channel 4/Value
//     PlcTask Inputs/GVL_iXlinker.EtherCAT_Master_EQxxxx.Beckhoff_EQ3xxx.Beckhoff_EQ3xxxEK1122.A_0009_EQ3204_0002_0021.WcState.WcState <-> WcState/WcState
//     PlcTask Inputs/GVL_iXlinker.EtherCAT_Master_EQxxxx.Beckhoff_EQ3xxx.Beckhoff_EQ3xxxEK1122.A_0009_EQ3204_0002_0021.WcState.InputToggle <-> WcState/InputToggle
//     PlcTask Inputs/GVL_iXlinker.EtherCAT_Master_EQxxxx.Beckhoff_EQ3xxx.Beckhoff_EQ3xxxEK1122.A_0009_EQ3204_0002_0021.InfoData.AdsAddr <-> InfoData/AdsAddr
//     PlcTask Inputs/GVL_iXlinker.EtherCAT_Master_EQxxxx.Beckhoff_EQ3xxx.Beckhoff_EQ3xxxEK1122.A_0009_EQ3204_0002_0021.InfoData.State <-> InfoData/State
//   PLC/PLC Instance <-> EtherCAT Master EQxxxx/Beckhoff EQ3xxx/Beckhoff EQ3xxxEK1122/A_0010(EQ3204-0002-0022)
//     PlcTask Inputs/GVL_iXlinker.EtherCAT_Master_EQxxxx.Beckhoff_EQ3xxx.Beckhoff_EQ3xxxEK1122.A_0010_EQ3204_0002_0022.RTD_RTDInputs_Channel_1.Status/Underrange <-> RTD RTDInputs Channel 1/Status/Underrange
//     PlcTask Inputs/GVL_iXlinker.EtherCAT_Master_EQxxxx.Beckhoff_EQ3xxx.Beckhoff_EQ3xxxEK1122.A_0010_EQ3204_0002_0022.RTD_RTDInputs_Channel_2.Status/Underrange <-> RTD RTDInputs Channel 2/Status/Underrange
//     PlcTask Inputs/GVL_iXlinker.EtherCAT_Master_EQxxxx.Beckhoff_EQ3xxx.Beckhoff_EQ3xxxEK1122.A_0010_EQ3204_0002_0022.RTD_RTDInputs_Channel_3.Status/Underrange <-> RTD RTDInputs Channel 3/Status/Underrange
//     PlcTask Inputs/GVL_iXlinker.EtherCAT_Master_EQxxxx.Beckhoff_EQ3xxx.Beckhoff_EQ3xxxEK1122.A_0010_EQ3204_0002_0022.RTD_RTDInputs_Channel_4.Status/Underrange <-> RTD RTDInputs Channel 4/Status/Underrange
//     PlcTask Inputs/GVL_iXlinker.EtherCAT_Master_EQxxxx.Beckhoff_EQ3xxx.Beckhoff_EQ3xxxEK1122.A_0010_EQ3204_0002_0022.RTD_RTDInputs_Channel_1.Status/Overrange <-> RTD RTDInputs Channel 1/Status/Overrange
//     PlcTask Inputs/GVL_iXlinker.EtherCAT_Master_EQxxxx.Beckhoff_EQ3xxx.Beckhoff_EQ3xxxEK1122.A_0010_EQ3204_0002_0022.RTD_RTDInputs_Channel_2.Status/Overrange <-> RTD RTDInputs Channel 2/Status/Overrange
//     PlcTask Inputs/GVL_iXlinker.EtherCAT_Master_EQxxxx.Beckhoff_EQ3xxx.Beckhoff_EQ3xxxEK1122.A_0010_EQ3204_0002_0022.RTD_RTDInputs_Channel_3.Status/Overrange <-> RTD RTDInputs Channel 3/Status/Overrange
//     PlcTask Inputs/GVL_iXlinker.EtherCAT_Master_EQxxxx.Beckhoff_EQ3xxx.Beckhoff_EQ3xxxEK1122.A_0010_EQ3204_0002_0022.RTD_RTDInputs_Channel_4.Status/Overrange <-> RTD RTDInputs Channel 4/Status/Overrange
//     PlcTask Inputs/GVL_iXlinker.EtherCAT_Master_EQxxxx.Beckhoff_EQ3xxx.Beckhoff_EQ3xxxEK1122.A_0010_EQ3204_0002_0022.RTD_RTDInputs_Channel_1.Status/Limit_1 <-> RTD RTDInputs Channel 1/Status/Limit 1
//     PlcTask Inputs/GVL_iXlinker.EtherCAT_Master_EQxxxx.Beckhoff_EQ3xxx.Beckhoff_EQ3xxxEK1122.A_0010_EQ3204_0002_0022.RTD_RTDInputs_Channel_1.Status/Limit_2 <-> RTD RTDInputs Channel 1/Status/Limit 2
//     PlcTask Inputs/GVL_iXlinker.EtherCAT_Master_EQxxxx.Beckhoff_EQ3xxx.Beckhoff_EQ3xxxEK1122.A_0010_EQ3204_0002_0022.RTD_RTDInputs_Channel_2.Status/Limit_1 <-> RTD RTDInputs Channel 2/Status/Limit 1
//     PlcTask Inputs/GVL_iXlinker.EtherCAT_Master_EQxxxx.Beckhoff_EQ3xxx.Beckhoff_EQ3xxxEK1122.A_0010_EQ3204_0002_0022.RTD_RTDInputs_Channel_2.Status/Limit_2 <-> RTD RTDInputs Channel 2/Status/Limit 2
//     PlcTask Inputs/GVL_iXlinker.EtherCAT_Master_EQxxxx.Beckhoff_EQ3xxx.Beckhoff_EQ3xxxEK1122.A_0010_EQ3204_0002_0022.RTD_RTDInputs_Channel_3.Status/Limit_1 <-> RTD RTDInputs Channel 3/Status/Limit 1
//     PlcTask Inputs/GVL_iXlinker.EtherCAT_Master_EQxxxx.Beckhoff_EQ3xxx.Beckhoff_EQ3xxxEK1122.A_0010_EQ3204_0002_0022.RTD_RTDInputs_Channel_3.Status/Limit_2 <-> RTD RTDInputs Channel 3/Status/Limit 2
//     PlcTask Inputs/GVL_iXlinker.EtherCAT_Master_EQxxxx.Beckhoff_EQ3xxx.Beckhoff_EQ3xxxEK1122.A_0010_EQ3204_0002_0022.RTD_RTDInputs_Channel_4.Status/Limit_1 <-> RTD RTDInputs Channel 4/Status/Limit 1
//     PlcTask Inputs/GVL_iXlinker.EtherCAT_Master_EQxxxx.Beckhoff_EQ3xxx.Beckhoff_EQ3xxxEK1122.A_0010_EQ3204_0002_0022.RTD_RTDInputs_Channel_4.Status/Limit_2 <-> RTD RTDInputs Channel 4/Status/Limit 2
//     PlcTask Inputs/GVL_iXlinker.EtherCAT_Master_EQxxxx.Beckhoff_EQ3xxx.Beckhoff_EQ3xxxEK1122.A_0010_EQ3204_0002_0022.RTD_RTDInputs_Channel_1.Status/Error <-> RTD RTDInputs Channel 1/Status/Error
//     PlcTask Inputs/GVL_iXlinker.EtherCAT_Master_EQxxxx.Beckhoff_EQ3xxx.Beckhoff_EQ3xxxEK1122.A_0010_EQ3204_0002_0022.RTD_RTDInputs_Channel_2.Status/Error <-> RTD RTDInputs Channel 2/Status/Error
//     PlcTask Inputs/GVL_iXlinker.EtherCAT_Master_EQxxxx.Beckhoff_EQ3xxx.Beckhoff_EQ3xxxEK1122.A_0010_EQ3204_0002_0022.RTD_RTDInputs_Channel_3.Status/Error <-> RTD RTDInputs Channel 3/Status/Error
//     PlcTask Inputs/GVL_iXlinker.EtherCAT_Master_EQxxxx.Beckhoff_EQ3xxx.Beckhoff_EQ3xxxEK1122.A_0010_EQ3204_0002_0022.RTD_RTDInputs_Channel_4.Status/Error <-> RTD RTDInputs Channel 4/Status/Error
//     PlcTask Inputs/GVL_iXlinker.EtherCAT_Master_EQxxxx.Beckhoff_EQ3xxx.Beckhoff_EQ3xxxEK1122.A_0010_EQ3204_0002_0022.RTD_RTDInputs_Channel_1.Status/TxPDO_State <-> RTD RTDInputs Channel 1/Status/TxPDO State
//     PlcTask Inputs/GVL_iXlinker.EtherCAT_Master_EQxxxx.Beckhoff_EQ3xxx.Beckhoff_EQ3xxxEK1122.A_0010_EQ3204_0002_0022.RTD_RTDInputs_Channel_2.Status/TxPDO_State <-> RTD RTDInputs Channel 2/Status/TxPDO State
//     PlcTask Inputs/GVL_iXlinker.EtherCAT_Master_EQxxxx.Beckhoff_EQ3xxx.Beckhoff_EQ3xxxEK1122.A_0010_EQ3204_0002_0022.RTD_RTDInputs_Channel_3.Status/TxPDO_State <-> RTD RTDInputs Channel 3/Status/TxPDO State
//     PlcTask Inputs/GVL_iXlinker.EtherCAT_Master_EQxxxx.Beckhoff_EQ3xxx.Beckhoff_EQ3xxxEK1122.A_0010_EQ3204_0002_0022.RTD_RTDInputs_Channel_4.Status/TxPDO_State <-> RTD RTDInputs Channel 4/Status/TxPDO State
//     PlcTask Inputs/GVL_iXlinker.EtherCAT_Master_EQxxxx.Beckhoff_EQ3xxx.Beckhoff_EQ3xxxEK1122.A_0010_EQ3204_0002_0022.RTD_RTDInputs_Channel_1.Status/TxPDO_Toggle <-> RTD RTDInputs Channel 1/Status/TxPDO Toggle
//     PlcTask Inputs/GVL_iXlinker.EtherCAT_Master_EQxxxx.Beckhoff_EQ3xxx.Beckhoff_EQ3xxxEK1122.A_0010_EQ3204_0002_0022.RTD_RTDInputs_Channel_2.Status/TxPDO_Toggle <-> RTD RTDInputs Channel 2/Status/TxPDO Toggle
//     PlcTask Inputs/GVL_iXlinker.EtherCAT_Master_EQxxxx.Beckhoff_EQ3xxx.Beckhoff_EQ3xxxEK1122.A_0010_EQ3204_0002_0022.RTD_RTDInputs_Channel_3.Status/TxPDO_Toggle <-> RTD RTDInputs Channel 3/Status/TxPDO Toggle
//     PlcTask Inputs/GVL_iXlinker.EtherCAT_Master_EQxxxx.Beckhoff_EQ3xxx.Beckhoff_EQ3xxxEK1122.A_0010_EQ3204_0002_0022.RTD_RTDInputs_Channel_4.Status/TxPDO_Toggle <-> RTD RTDInputs Channel 4/Status/TxPDO Toggle
//     PlcTask Inputs/GVL_iXlinker.EtherCAT_Master_EQxxxx.Beckhoff_EQ3xxx.Beckhoff_EQ3xxxEK1122.A_0010_EQ3204_0002_0022.RTD_RTDInputs_Channel_1.Value <-> RTD RTDInputs Channel 1/Value
//     PlcTask Inputs/GVL_iXlinker.EtherCAT_Master_EQxxxx.Beckhoff_EQ3xxx.Beckhoff_EQ3xxxEK1122.A_0010_EQ3204_0002_0022.RTD_RTDInputs_Channel_2.Value <-> RTD RTDInputs Channel 2/Value
//     PlcTask Inputs/GVL_iXlinker.EtherCAT_Master_EQxxxx.Beckhoff_EQ3xxx.Beckhoff_EQ3xxxEK1122.A_0010_EQ3204_0002_0022.RTD_RTDInputs_Channel_3.Value <-> RTD RTDInputs Channel 3/Value
//     PlcTask Inputs/GVL_iXlinker.EtherCAT_Master_EQxxxx.Beckhoff_EQ3xxx.Beckhoff_EQ3xxxEK1122.A_0010_EQ3204_0002_0022.RTD_RTDInputs_Channel_4.Value <-> RTD RTDInputs Channel 4/Value
//     PlcTask Inputs/GVL_iXlinker.EtherCAT_Master_EQxxxx.Beckhoff_EQ3xxx.Beckhoff_EQ3xxxEK1122.A_0010_EQ3204_0002_0022.WcState.WcState <-> WcState/WcState
//     PlcTask Inputs/GVL_iXlinker.EtherCAT_Master_EQxxxx.Beckhoff_EQ3xxx.Beckhoff_EQ3xxxEK1122.A_0010_EQ3204_0002_0022.WcState.InputToggle <-> WcState/InputToggle
//     PlcTask Inputs/GVL_iXlinker.EtherCAT_Master_EQxxxx.Beckhoff_EQ3xxx.Beckhoff_EQ3xxxEK1122.A_0010_EQ3204_0002_0022.InfoData.AdsAddr <-> InfoData/AdsAddr
//     PlcTask Inputs/GVL_iXlinker.EtherCAT_Master_EQxxxx.Beckhoff_EQ3xxx.Beckhoff_EQ3xxxEK1122.A_0010_EQ3204_0002_0022.InfoData.State <-> InfoData/State
//   PLC/PLC Instance <-> EtherCAT Master EQxxxx/Beckhoff EQ3xxx/Beckhoff EQ3xxxEK1122/A_0011(EQ3314-0002-0016)
//     PlcTask Inputs/GVL_iXlinker.EtherCAT_Master_EQxxxx.Beckhoff_EQ3xxx.Beckhoff_EQ3xxxEK1122.A_0011_EQ3314_0002_0016.TC_TCInputs_Channel_1.Status/Underrange <-> TC TCInputs Channel 1/Status/Underrange
//     PlcTask Inputs/GVL_iXlinker.EtherCAT_Master_EQxxxx.Beckhoff_EQ3xxx.Beckhoff_EQ3xxxEK1122.A_0011_EQ3314_0002_0016.TC_TCInputs_Channel_2.Status/Underrange <-> TC TCInputs Channel 2/Status/Underrange
//     PlcTask Inputs/GVL_iXlinker.EtherCAT_Master_EQxxxx.Beckhoff_EQ3xxx.Beckhoff_EQ3xxxEK1122.A_0011_EQ3314_0002_0016.TC_TCInputs_Channel_3.Status/Underrange <-> TC TCInputs Channel 3/Status/Underrange
//     PlcTask Inputs/GVL_iXlinker.EtherCAT_Master_EQxxxx.Beckhoff_EQ3xxx.Beckhoff_EQ3xxxEK1122.A_0011_EQ3314_0002_0016.TC_TCInputs_Channel_4.Status/Underrange <-> TC TCInputs Channel 4/Status/Underrange
//     PlcTask Inputs/GVL_iXlinker.EtherCAT_Master_EQxxxx.Beckhoff_EQ3xxx.Beckhoff_EQ3xxxEK1122.A_0011_EQ3314_0002_0016.TC_TCInputs_Channel_1.Status/Overrange <-> TC TCInputs Channel 1/Status/Overrange
//     PlcTask Inputs/GVL_iXlinker.EtherCAT_Master_EQxxxx.Beckhoff_EQ3xxx.Beckhoff_EQ3xxxEK1122.A_0011_EQ3314_0002_0016.TC_TCInputs_Channel_2.Status/Overrange <-> TC TCInputs Channel 2/Status/Overrange
//     PlcTask Inputs/GVL_iXlinker.EtherCAT_Master_EQxxxx.Beckhoff_EQ3xxx.Beckhoff_EQ3xxxEK1122.A_0011_EQ3314_0002_0016.TC_TCInputs_Channel_3.Status/Overrange <-> TC TCInputs Channel 3/Status/Overrange
//     PlcTask Inputs/GVL_iXlinker.EtherCAT_Master_EQxxxx.Beckhoff_EQ3xxx.Beckhoff_EQ3xxxEK1122.A_0011_EQ3314_0002_0016.TC_TCInputs_Channel_4.Status/Overrange <-> TC TCInputs Channel 4/Status/Overrange
//     PlcTask Inputs/GVL_iXlinker.EtherCAT_Master_EQxxxx.Beckhoff_EQ3xxx.Beckhoff_EQ3xxxEK1122.A_0011_EQ3314_0002_0016.TC_TCInputs_Channel_1.Status/Limit_1 <-> TC TCInputs Channel 1/Status/Limit 1
//     PlcTask Inputs/GVL_iXlinker.EtherCAT_Master_EQxxxx.Beckhoff_EQ3xxx.Beckhoff_EQ3xxxEK1122.A_0011_EQ3314_0002_0016.TC_TCInputs_Channel_1.Status/Limit_2 <-> TC TCInputs Channel 1/Status/Limit 2
//     PlcTask Inputs/GVL_iXlinker.EtherCAT_Master_EQxxxx.Beckhoff_EQ3xxx.Beckhoff_EQ3xxxEK1122.A_0011_EQ3314_0002_0016.TC_TCInputs_Channel_2.Status/Limit_1 <-> TC TCInputs Channel 2/Status/Limit 1
//     PlcTask Inputs/GVL_iXlinker.EtherCAT_Master_EQxxxx.Beckhoff_EQ3xxx.Beckhoff_EQ3xxxEK1122.A_0011_EQ3314_0002_0016.TC_TCInputs_Channel_2.Status/Limit_2 <-> TC TCInputs Channel 2/Status/Limit 2
//     PlcTask Inputs/GVL_iXlinker.EtherCAT_Master_EQxxxx.Beckhoff_EQ3xxx.Beckhoff_EQ3xxxEK1122.A_0011_EQ3314_0002_0016.TC_TCInputs_Channel_3.Status/Limit_1 <-> TC TCInputs Channel 3/Status/Limit 1
//     PlcTask Inputs/GVL_iXlinker.EtherCAT_Master_EQxxxx.Beckhoff_EQ3xxx.Beckhoff_EQ3xxxEK1122.A_0011_EQ3314_0002_0016.TC_TCInputs_Channel_3.Status/Limit_2 <-> TC TCInputs Channel 3/Status/Limit 2
//     PlcTask Inputs/GVL_iXlinker.EtherCAT_Master_EQxxxx.Beckhoff_EQ3xxx.Beckhoff_EQ3xxxEK1122.A_0011_EQ3314_0002_0016.TC_TCInputs_Channel_4.Status/Limit_1 <-> TC TCInputs Channel 4/Status/Limit 1
//     PlcTask Inputs/GVL_iXlinker.EtherCAT_Master_EQxxxx.Beckhoff_EQ3xxx.Beckhoff_EQ3xxxEK1122.A_0011_EQ3314_0002_0016.TC_TCInputs_Channel_4.Status/Limit_2 <-> TC TCInputs Channel 4/Status/Limit 2
//     PlcTask Inputs/GVL_iXlinker.EtherCAT_Master_EQxxxx.Beckhoff_EQ3xxx.Beckhoff_EQ3xxxEK1122.A_0011_EQ3314_0002_0016.TC_TCInputs_Channel_1.Status/Error <-> TC TCInputs Channel 1/Status/Error
//     PlcTask Inputs/GVL_iXlinker.EtherCAT_Master_EQxxxx.Beckhoff_EQ3xxx.Beckhoff_EQ3xxxEK1122.A_0011_EQ3314_0002_0016.TC_TCInputs_Channel_2.Status/Error <-> TC TCInputs Channel 2/Status/Error
//     PlcTask Inputs/GVL_iXlinker.EtherCAT_Master_EQxxxx.Beckhoff_EQ3xxx.Beckhoff_EQ3xxxEK1122.A_0011_EQ3314_0002_0016.TC_TCInputs_Channel_3.Status/Error <-> TC TCInputs Channel 3/Status/Error
//     PlcTask Inputs/GVL_iXlinker.EtherCAT_Master_EQxxxx.Beckhoff_EQ3xxx.Beckhoff_EQ3xxxEK1122.A_0011_EQ3314_0002_0016.TC_TCInputs_Channel_4.Status/Error <-> TC TCInputs Channel 4/Status/Error
//     PlcTask Inputs/GVL_iXlinker.EtherCAT_Master_EQxxxx.Beckhoff_EQ3xxx.Beckhoff_EQ3xxxEK1122.A_0011_EQ3314_0002_0016.TC_TCInputs_Channel_1.Status/Sync_error <-> TC TCInputs Channel 1/Status/Sync error
//     PlcTask Inputs/GVL_iXlinker.EtherCAT_Master_EQxxxx.Beckhoff_EQ3xxx.Beckhoff_EQ3xxxEK1122.A_0011_EQ3314_0002_0016.TC_TCInputs_Channel_2.Status/Sync_error <-> TC TCInputs Channel 2/Status/Sync error
//     PlcTask Inputs/GVL_iXlinker.EtherCAT_Master_EQxxxx.Beckhoff_EQ3xxx.Beckhoff_EQ3xxxEK1122.A_0011_EQ3314_0002_0016.TC_TCInputs_Channel_3.Status/Sync_error <-> TC TCInputs Channel 3/Status/Sync error
//     PlcTask Inputs/GVL_iXlinker.EtherCAT_Master_EQxxxx.Beckhoff_EQ3xxx.Beckhoff_EQ3xxxEK1122.A_0011_EQ3314_0002_0016.TC_TCInputs_Channel_4.Status/Sync_error <-> TC TCInputs Channel 4/Status/Sync error
//     PlcTask Inputs/GVL_iXlinker.EtherCAT_Master_EQxxxx.Beckhoff_EQ3xxx.Beckhoff_EQ3xxxEK1122.A_0011_EQ3314_0002_0016.TC_TCInputs_Channel_1.Status/TxPDO_State <-> TC TCInputs Channel 1/Status/TxPDO State
//     PlcTask Inputs/GVL_iXlinker.EtherCAT_Master_EQxxxx.Beckhoff_EQ3xxx.Beckhoff_EQ3xxxEK1122.A_0011_EQ3314_0002_0016.TC_TCInputs_Channel_2.Status/TxPDO_State <-> TC TCInputs Channel 2/Status/TxPDO State
//     PlcTask Inputs/GVL_iXlinker.EtherCAT_Master_EQxxxx.Beckhoff_EQ3xxx.Beckhoff_EQ3xxxEK1122.A_0011_EQ3314_0002_0016.TC_TCInputs_Channel_3.Status/TxPDO_State <-> TC TCInputs Channel 3/Status/TxPDO State
//     PlcTask Inputs/GVL_iXlinker.EtherCAT_Master_EQxxxx.Beckhoff_EQ3xxx.Beckhoff_EQ3xxxEK1122.A_0011_EQ3314_0002_0016.TC_TCInputs_Channel_4.Status/TxPDO_State <-> TC TCInputs Channel 4/Status/TxPDO State
//     PlcTask Inputs/GVL_iXlinker.EtherCAT_Master_EQxxxx.Beckhoff_EQ3xxx.Beckhoff_EQ3xxxEK1122.A_0011_EQ3314_0002_0016.TC_TCInputs_Channel_1.Status/TxPDO_Toggle <-> TC TCInputs Channel 1/Status/TxPDO Toggle
//     PlcTask Inputs/GVL_iXlinker.EtherCAT_Master_EQxxxx.Beckhoff_EQ3xxx.Beckhoff_EQ3xxxEK1122.A_0011_EQ3314_0002_0016.TC_TCInputs_Channel_2.Status/TxPDO_Toggle <-> TC TCInputs Channel 2/Status/TxPDO Toggle
//     PlcTask Inputs/GVL_iXlinker.EtherCAT_Master_EQxxxx.Beckhoff_EQ3xxx.Beckhoff_EQ3xxxEK1122.A_0011_EQ3314_0002_0016.TC_TCInputs_Channel_3.Status/TxPDO_Toggle <-> TC TCInputs Channel 3/Status/TxPDO Toggle
//     PlcTask Inputs/GVL_iXlinker.EtherCAT_Master_EQxxxx.Beckhoff_EQ3xxx.Beckhoff_EQ3xxxEK1122.A_0011_EQ3314_0002_0016.TC_TCInputs_Channel_4.Status/TxPDO_Toggle <-> TC TCInputs Channel 4/Status/TxPDO Toggle
//     PlcTask Inputs/GVL_iXlinker.EtherCAT_Master_EQxxxx.Beckhoff_EQ3xxx.Beckhoff_EQ3xxxEK1122.A_0011_EQ3314_0002_0016.TC_TCInputs_Channel_1.Value <-> TC TCInputs Channel 1/Value
//     PlcTask Inputs/GVL_iXlinker.EtherCAT_Master_EQxxxx.Beckhoff_EQ3xxx.Beckhoff_EQ3xxxEK1122.A_0011_EQ3314_0002_0016.TC_TCInputs_Channel_2.Value <-> TC TCInputs Channel 2/Value
//     PlcTask Inputs/GVL_iXlinker.EtherCAT_Master_EQxxxx.Beckhoff_EQ3xxx.Beckhoff_EQ3xxxEK1122.A_0011_EQ3314_0002_0016.TC_TCInputs_Channel_3.Value <-> TC TCInputs Channel 3/Value
//     PlcTask Inputs/GVL_iXlinker.EtherCAT_Master_EQxxxx.Beckhoff_EQ3xxx.Beckhoff_EQ3xxxEK1122.A_0011_EQ3314_0002_0016.TC_TCInputs_Channel_4.Value <-> TC TCInputs Channel 4/Value
//     PlcTask Inputs/GVL_iXlinker.EtherCAT_Master_EQxxxx.Beckhoff_EQ3xxx.Beckhoff_EQ3xxxEK1122.A_0011_EQ3314_0002_0016.WcState.WcState <-> WcState/WcState
//     PlcTask Inputs/GVL_iXlinker.EtherCAT_Master_EQxxxx.Beckhoff_EQ3xxx.Beckhoff_EQ3xxxEK1122.A_0011_EQ3314_0002_0016.WcState.InputToggle <-> WcState/InputToggle
//     PlcTask Inputs/GVL_iXlinker.EtherCAT_Master_EQxxxx.Beckhoff_EQ3xxx.Beckhoff_EQ3xxxEK1122.A_0011_EQ3314_0002_0016.InfoData.AdsAddr <-> InfoData/AdsAddr
//     PlcTask Inputs/GVL_iXlinker.EtherCAT_Master_EQxxxx.Beckhoff_EQ3xxx.Beckhoff_EQ3xxxEK1122.A_0011_EQ3314_0002_0016.InfoData.State <-> InfoData/State
//   PLC/PLC Instance <-> EtherCAT Master EQxxxx/Beckhoff EQ3xxx/Beckhoff EQ3xxxEK1122/A_0012(EQ3314-0002-0017)
//     PlcTask Inputs/GVL_iXlinker.EtherCAT_Master_EQxxxx.Beckhoff_EQ3xxx.Beckhoff_EQ3xxxEK1122.A_0012_EQ3314_0002_0017.TC_TCInputs_Channel_1.Status/Underrange <-> TC TCInputs Channel 1/Status/Underrange
//     PlcTask Inputs/GVL_iXlinker.EtherCAT_Master_EQxxxx.Beckhoff_EQ3xxx.Beckhoff_EQ3xxxEK1122.A_0012_EQ3314_0002_0017.TC_TCInputs_Channel_2.Status/Underrange <-> TC TCInputs Channel 2/Status/Underrange
//     PlcTask Inputs/GVL_iXlinker.EtherCAT_Master_EQxxxx.Beckhoff_EQ3xxx.Beckhoff_EQ3xxxEK1122.A_0012_EQ3314_0002_0017.TC_TCInputs_Channel_3.Status/Underrange <-> TC TCInputs Channel 3/Status/Underrange
//     PlcTask Inputs/GVL_iXlinker.EtherCAT_Master_EQxxxx.Beckhoff_EQ3xxx.Beckhoff_EQ3xxxEK1122.A_0012_EQ3314_0002_0017.TC_TCInputs_Channel_4.Status/Underrange <-> TC TCInputs Channel 4/Status/Underrange
//     PlcTask Inputs/GVL_iXlinker.EtherCAT_Master_EQxxxx.Beckhoff_EQ3xxx.Beckhoff_EQ3xxxEK1122.A_0012_EQ3314_0002_0017.TC_TCInputs_Channel_1.Status/Overrange <-> TC TCInputs Channel 1/Status/Overrange
//     PlcTask Inputs/GVL_iXlinker.EtherCAT_Master_EQxxxx.Beckhoff_EQ3xxx.Beckhoff_EQ3xxxEK1122.A_0012_EQ3314_0002_0017.TC_TCInputs_Channel_2.Status/Overrange <-> TC TCInputs Channel 2/Status/Overrange
//     PlcTask Inputs/GVL_iXlinker.EtherCAT_Master_EQxxxx.Beckhoff_EQ3xxx.Beckhoff_EQ3xxxEK1122.A_0012_EQ3314_0002_0017.TC_TCInputs_Channel_3.Status/Overrange <-> TC TCInputs Channel 3/Status/Overrange
//     PlcTask Inputs/GVL_iXlinker.EtherCAT_Master_EQxxxx.Beckhoff_EQ3xxx.Beckhoff_EQ3xxxEK1122.A_0012_EQ3314_0002_0017.TC_TCInputs_Channel_4.Status/Overrange <-> TC TCInputs Channel 4/Status/Overrange
//     PlcTask Inputs/GVL_iXlinker.EtherCAT_Master_EQxxxx.Beckhoff_EQ3xxx.Beckhoff_EQ3xxxEK1122.A_0012_EQ3314_0002_0017.TC_TCInputs_Channel_1.Status/Limit_1 <-> TC TCInputs Channel 1/Status/Limit 1
//     PlcTask Inputs/GVL_iXlinker.EtherCAT_Master_EQxxxx.Beckhoff_EQ3xxx.Beckhoff_EQ3xxxEK1122.A_0012_EQ3314_0002_0017.TC_TCInputs_Channel_1.Status/Limit_2 <-> TC TCInputs Channel 1/Status/Limit 2
//     PlcTask Inputs/GVL_iXlinker.EtherCAT_Master_EQxxxx.Beckhoff_EQ3xxx.Beckhoff_EQ3xxxEK1122.A_0012_EQ3314_0002_0017.TC_TCInputs_Channel_2.Status/Limit_1 <-> TC TCInputs Channel 2/Status/Limit 1
//     PlcTask Inputs/GVL_iXlinker.EtherCAT_Master_EQxxxx.Beckhoff_EQ3xxx.Beckhoff_EQ3xxxEK1122.A_0012_EQ3314_0002_0017.TC_TCInputs_Channel_2.Status/Limit_2 <-> TC TCInputs Channel 2/Status/Limit 2
//     PlcTask Inputs/GVL_iXlinker.EtherCAT_Master_EQxxxx.Beckhoff_EQ3xxx.Beckhoff_EQ3xxxEK1122.A_0012_EQ3314_0002_0017.TC_TCInputs_Channel_3.Status/Limit_1 <-> TC TCInputs Channel 3/Status/Limit 1
//     PlcTask Inputs/GVL_iXlinker.EtherCAT_Master_EQxxxx.Beckhoff_EQ3xxx.Beckhoff_EQ3xxxEK1122.A_0012_EQ3314_0002_0017.TC_TCInputs_Channel_3.Status/Limit_2 <-> TC TCInputs Channel 3/Status/Limit 2
//     PlcTask Inputs/GVL_iXlinker.EtherCAT_Master_EQxxxx.Beckhoff_EQ3xxx.Beckhoff_EQ3xxxEK1122.A_0012_EQ3314_0002_0017.TC_TCInputs_Channel_4.Status/Limit_1 <-> TC TCInputs Channel 4/Status/Limit 1
//     PlcTask Inputs/GVL_iXlinker.EtherCAT_Master_EQxxxx.Beckhoff_EQ3xxx.Beckhoff_EQ3xxxEK1122.A_0012_EQ3314_0002_0017.TC_TCInputs_Channel_4.Status/Limit_2 <-> TC TCInputs Channel 4/Status/Limit 2
//     PlcTask Inputs/GVL_iXlinker.EtherCAT_Master_EQxxxx.Beckhoff_EQ3xxx.Beckhoff_EQ3xxxEK1122.A_0012_EQ3314_0002_0017.TC_TCInputs_Channel_1.Status/Error <-> TC TCInputs Channel 1/Status/Error
//     PlcTask Inputs/GVL_iXlinker.EtherCAT_Master_EQxxxx.Beckhoff_EQ3xxx.Beckhoff_EQ3xxxEK1122.A_0012_EQ3314_0002_0017.TC_TCInputs_Channel_2.Status/Error <-> TC TCInputs Channel 2/Status/Error
//     PlcTask Inputs/GVL_iXlinker.EtherCAT_Master_EQxxxx.Beckhoff_EQ3xxx.Beckhoff_EQ3xxxEK1122.A_0012_EQ3314_0002_0017.TC_TCInputs_Channel_3.Status/Error <-> TC TCInputs Channel 3/Status/Error
//     PlcTask Inputs/GVL_iXlinker.EtherCAT_Master_EQxxxx.Beckhoff_EQ3xxx.Beckhoff_EQ3xxxEK1122.A_0012_EQ3314_0002_0017.TC_TCInputs_Channel_4.Status/Error <-> TC TCInputs Channel 4/Status/Error
//     PlcTask Inputs/GVL_iXlinker.EtherCAT_Master_EQxxxx.Beckhoff_EQ3xxx.Beckhoff_EQ3xxxEK1122.A_0012_EQ3314_0002_0017.TC_TCInputs_Channel_1.Status/Sync_error <-> TC TCInputs Channel 1/Status/Sync error
//     PlcTask Inputs/GVL_iXlinker.EtherCAT_Master_EQxxxx.Beckhoff_EQ3xxx.Beckhoff_EQ3xxxEK1122.A_0012_EQ3314_0002_0017.TC_TCInputs_Channel_2.Status/Sync_error <-> TC TCInputs Channel 2/Status/Sync error
//     PlcTask Inputs/GVL_iXlinker.EtherCAT_Master_EQxxxx.Beckhoff_EQ3xxx.Beckhoff_EQ3xxxEK1122.A_0012_EQ3314_0002_0017.TC_TCInputs_Channel_3.Status/Sync_error <-> TC TCInputs Channel 3/Status/Sync error
//     PlcTask Inputs/GVL_iXlinker.EtherCAT_Master_EQxxxx.Beckhoff_EQ3xxx.Beckhoff_EQ3xxxEK1122.A_0012_EQ3314_0002_0017.TC_TCInputs_Channel_4.Status/Sync_error <-> TC TCInputs Channel 4/Status/Sync error
//     PlcTask Inputs/GVL_iXlinker.EtherCAT_Master_EQxxxx.Beckhoff_EQ3xxx.Beckhoff_EQ3xxxEK1122.A_0012_EQ3314_0002_0017.TC_TCInputs_Channel_1.Status/TxPDO_State <-> TC TCInputs Channel 1/Status/TxPDO State
//     PlcTask Inputs/GVL_iXlinker.EtherCAT_Master_EQxxxx.Beckhoff_EQ3xxx.Beckhoff_EQ3xxxEK1122.A_0012_EQ3314_0002_0017.TC_TCInputs_Channel_2.Status/TxPDO_State <-> TC TCInputs Channel 2/Status/TxPDO State
//     PlcTask Inputs/GVL_iXlinker.EtherCAT_Master_EQxxxx.Beckhoff_EQ3xxx.Beckhoff_EQ3xxxEK1122.A_0012_EQ3314_0002_0017.TC_TCInputs_Channel_3.Status/TxPDO_State <-> TC TCInputs Channel 3/Status/TxPDO State
//     PlcTask Inputs/GVL_iXlinker.EtherCAT_Master_EQxxxx.Beckhoff_EQ3xxx.Beckhoff_EQ3xxxEK1122.A_0012_EQ3314_0002_0017.TC_TCInputs_Channel_4.Status/TxPDO_State <-> TC TCInputs Channel 4/Status/TxPDO State
//     PlcTask Inputs/GVL_iXlinker.EtherCAT_Master_EQxxxx.Beckhoff_EQ3xxx.Beckhoff_EQ3xxxEK1122.A_0012_EQ3314_0002_0017.TC_TCInputs_Channel_1.Status/TxPDO_Toggle <-> TC TCInputs Channel 1/Status/TxPDO Toggle
//     PlcTask Inputs/GVL_iXlinker.EtherCAT_Master_EQxxxx.Beckhoff_EQ3xxx.Beckhoff_EQ3xxxEK1122.A_0012_EQ3314_0002_0017.TC_TCInputs_Channel_2.Status/TxPDO_Toggle <-> TC TCInputs Channel 2/Status/TxPDO Toggle
//     PlcTask Inputs/GVL_iXlinker.EtherCAT_Master_EQxxxx.Beckhoff_EQ3xxx.Beckhoff_EQ3xxxEK1122.A_0012_EQ3314_0002_0017.TC_TCInputs_Channel_3.Status/TxPDO_Toggle <-> TC TCInputs Channel 3/Status/TxPDO Toggle
//     PlcTask Inputs/GVL_iXlinker.EtherCAT_Master_EQxxxx.Beckhoff_EQ3xxx.Beckhoff_EQ3xxxEK1122.A_0012_EQ3314_0002_0017.TC_TCInputs_Channel_4.Status/TxPDO_Toggle <-> TC TCInputs Channel 4/Status/TxPDO Toggle
//     PlcTask Inputs/GVL_iXlinker.EtherCAT_Master_EQxxxx.Beckhoff_EQ3xxx.Beckhoff_EQ3xxxEK1122.A_0012_EQ3314_0002_0017.TC_TCInputs_Channel_1.Value <-> TC TCInputs Channel 1/Value
//     PlcTask Inputs/GVL_iXlinker.EtherCAT_Master_EQxxxx.Beckhoff_EQ3xxx.Beckhoff_EQ3xxxEK1122.A_0012_EQ3314_0002_0017.TC_TCInputs_Channel_2.Value <-> TC TCInputs Channel 2/Value
//     PlcTask Inputs/GVL_iXlinker.EtherCAT_Master_EQxxxx.Beckhoff_EQ3xxx.Beckhoff_EQ3xxxEK1122.A_0012_EQ3314_0002_0017.TC_TCInputs_Channel_3.Value <-> TC TCInputs Channel 3/Value
//     PlcTask Inputs/GVL_iXlinker.EtherCAT_Master_EQxxxx.Beckhoff_EQ3xxx.Beckhoff_EQ3xxxEK1122.A_0012_EQ3314_0002_0017.TC_TCInputs_Channel_4.Value <-> TC TCInputs Channel 4/Value
//     PlcTask Inputs/GVL_iXlinker.EtherCAT_Master_EQxxxx.Beckhoff_EQ3xxx.Beckhoff_EQ3xxxEK1122.A_0012_EQ3314_0002_0017.WcState.WcState <-> WcState/WcState
//     PlcTask Inputs/GVL_iXlinker.EtherCAT_Master_EQxxxx.Beckhoff_EQ3xxx.Beckhoff_EQ3xxxEK1122.A_0012_EQ3314_0002_0017.WcState.InputToggle <-> WcState/InputToggle
//     PlcTask Inputs/GVL_iXlinker.EtherCAT_Master_EQxxxx.Beckhoff_EQ3xxx.Beckhoff_EQ3xxxEK1122.A_0012_EQ3314_0002_0017.InfoData.AdsAddr <-> InfoData/AdsAddr
//     PlcTask Inputs/GVL_iXlinker.EtherCAT_Master_EQxxxx.Beckhoff_EQ3xxx.Beckhoff_EQ3xxxEK1122.A_0012_EQ3314_0002_0017.InfoData.State <-> InfoData/State
//   PLC/PLC Instance <-> EtherCAT Master EQxxxx/Beckhoff EQ3xxx/Beckhoff EQ3xxxEK1122/A_0013(EQ3314-0002-0021)
//     PlcTask Inputs/GVL_iXlinker.EtherCAT_Master_EQxxxx.Beckhoff_EQ3xxx.Beckhoff_EQ3xxxEK1122.A_0013_EQ3314_0002_0021.TC_TCInputs_Channel_1.Status/Underrange <-> TC TCInputs Channel 1/Status/Underrange
//     PlcTask Inputs/GVL_iXlinker.EtherCAT_Master_EQxxxx.Beckhoff_EQ3xxx.Beckhoff_EQ3xxxEK1122.A_0013_EQ3314_0002_0021.TC_TCInputs_Channel_2.Status/Underrange <-> TC TCInputs Channel 2/Status/Underrange
//     PlcTask Inputs/GVL_iXlinker.EtherCAT_Master_EQxxxx.Beckhoff_EQ3xxx.Beckhoff_EQ3xxxEK1122.A_0013_EQ3314_0002_0021.TC_TCInputs_Channel_3.Status/Underrange <-> TC TCInputs Channel 3/Status/Underrange
//     PlcTask Inputs/GVL_iXlinker.EtherCAT_Master_EQxxxx.Beckhoff_EQ3xxx.Beckhoff_EQ3xxxEK1122.A_0013_EQ3314_0002_0021.TC_TCInputs_Channel_4.Status/Underrange <-> TC TCInputs Channel 4/Status/Underrange
//     PlcTask Inputs/GVL_iXlinker.EtherCAT_Master_EQxxxx.Beckhoff_EQ3xxx.Beckhoff_EQ3xxxEK1122.A_0013_EQ3314_0002_0021.TC_TCInputs_Channel_1.Status/Overrange <-> TC TCInputs Channel 1/Status/Overrange
//     PlcTask Inputs/GVL_iXlinker.EtherCAT_Master_EQxxxx.Beckhoff_EQ3xxx.Beckhoff_EQ3xxxEK1122.A_0013_EQ3314_0002_0021.TC_TCInputs_Channel_2.Status/Overrange <-> TC TCInputs Channel 2/Status/Overrange
//     PlcTask Inputs/GVL_iXlinker.EtherCAT_Master_EQxxxx.Beckhoff_EQ3xxx.Beckhoff_EQ3xxxEK1122.A_0013_EQ3314_0002_0021.TC_TCInputs_Channel_3.Status/Overrange <-> TC TCInputs Channel 3/Status/Overrange
//     PlcTask Inputs/GVL_iXlinker.EtherCAT_Master_EQxxxx.Beckhoff_EQ3xxx.Beckhoff_EQ3xxxEK1122.A_0013_EQ3314_0002_0021.TC_TCInputs_Channel_4.Status/Overrange <-> TC TCInputs Channel 4/Status/Overrange
//     PlcTask Inputs/GVL_iXlinker.EtherCAT_Master_EQxxxx.Beckhoff_EQ3xxx.Beckhoff_EQ3xxxEK1122.A_0013_EQ3314_0002_0021.TC_TCInputs_Channel_1.Status/Limit_1 <-> TC TCInputs Channel 1/Status/Limit 1
//     PlcTask Inputs/GVL_iXlinker.EtherCAT_Master_EQxxxx.Beckhoff_EQ3xxx.Beckhoff_EQ3xxxEK1122.A_0013_EQ3314_0002_0021.TC_TCInputs_Channel_1.Status/Limit_2 <-> TC TCInputs Channel 1/Status/Limit 2
//     PlcTask Inputs/GVL_iXlinker.EtherCAT_Master_EQxxxx.Beckhoff_EQ3xxx.Beckhoff_EQ3xxxEK1122.A_0013_EQ3314_0002_0021.TC_TCInputs_Channel_2.Status/Limit_1 <-> TC TCInputs Channel 2/Status/Limit 1
//     PlcTask Inputs/GVL_iXlinker.EtherCAT_Master_EQxxxx.Beckhoff_EQ3xxx.Beckhoff_EQ3xxxEK1122.A_0013_EQ3314_0002_0021.TC_TCInputs_Channel_2.Status/Limit_2 <-> TC TCInputs Channel 2/Status/Limit 2
//     PlcTask Inputs/GVL_iXlinker.EtherCAT_Master_EQxxxx.Beckhoff_EQ3xxx.Beckhoff_EQ3xxxEK1122.A_0013_EQ3314_0002_0021.TC_TCInputs_Channel_3.Status/Limit_1 <-> TC TCInputs Channel 3/Status/Limit 1
//     PlcTask Inputs/GVL_iXlinker.EtherCAT_Master_EQxxxx.Beckhoff_EQ3xxx.Beckhoff_EQ3xxxEK1122.A_0013_EQ3314_0002_0021.TC_TCInputs_Channel_3.Status/Limit_2 <-> TC TCInputs Channel 3/Status/Limit 2
//     PlcTask Inputs/GVL_iXlinker.EtherCAT_Master_EQxxxx.Beckhoff_EQ3xxx.Beckhoff_EQ3xxxEK1122.A_0013_EQ3314_0002_0021.TC_TCInputs_Channel_4.Status/Limit_1 <-> TC TCInputs Channel 4/Status/Limit 1
//     PlcTask Inputs/GVL_iXlinker.EtherCAT_Master_EQxxxx.Beckhoff_EQ3xxx.Beckhoff_EQ3xxxEK1122.A_0013_EQ3314_0002_0021.TC_TCInputs_Channel_4.Status/Limit_2 <-> TC TCInputs Channel 4/Status/Limit 2
//     PlcTask Inputs/GVL_iXlinker.EtherCAT_Master_EQxxxx.Beckhoff_EQ3xxx.Beckhoff_EQ3xxxEK1122.A_0013_EQ3314_0002_0021.TC_TCInputs_Channel_1.Status/Error <-> TC TCInputs Channel 1/Status/Error
//     PlcTask Inputs/GVL_iXlinker.EtherCAT_Master_EQxxxx.Beckhoff_EQ3xxx.Beckhoff_EQ3xxxEK1122.A_0013_EQ3314_0002_0021.TC_TCInputs_Channel_2.Status/Error <-> TC TCInputs Channel 2/Status/Error
//     PlcTask Inputs/GVL_iXlinker.EtherCAT_Master_EQxxxx.Beckhoff_EQ3xxx.Beckhoff_EQ3xxxEK1122.A_0013_EQ3314_0002_0021.TC_TCInputs_Channel_3.Status/Error <-> TC TCInputs Channel 3/Status/Error
//     PlcTask Inputs/GVL_iXlinker.EtherCAT_Master_EQxxxx.Beckhoff_EQ3xxx.Beckhoff_EQ3xxxEK1122.A_0013_EQ3314_0002_0021.TC_TCInputs_Channel_4.Status/Error <-> TC TCInputs Channel 4/Status/Error
//     PlcTask Inputs/GVL_iXlinker.EtherCAT_Master_EQxxxx.Beckhoff_EQ3xxx.Beckhoff_EQ3xxxEK1122.A_0013_EQ3314_0002_0021.TC_TCInputs_Channel_1.Status/Sync_error <-> TC TCInputs Channel 1/Status/Sync error
//     PlcTask Inputs/GVL_iXlinker.EtherCAT_Master_EQxxxx.Beckhoff_EQ3xxx.Beckhoff_EQ3xxxEK1122.A_0013_EQ3314_0002_0021.TC_TCInputs_Channel_2.Status/Sync_error <-> TC TCInputs Channel 2/Status/Sync error
//     PlcTask Inputs/GVL_iXlinker.EtherCAT_Master_EQxxxx.Beckhoff_EQ3xxx.Beckhoff_EQ3xxxEK1122.A_0013_EQ3314_0002_0021.TC_TCInputs_Channel_3.Status/Sync_error <-> TC TCInputs Channel 3/Status/Sync error
//     PlcTask Inputs/GVL_iXlinker.EtherCAT_Master_EQxxxx.Beckhoff_EQ3xxx.Beckhoff_EQ3xxxEK1122.A_0013_EQ3314_0002_0021.TC_TCInputs_Channel_4.Status/Sync_error <-> TC TCInputs Channel 4/Status/Sync error
//     PlcTask Inputs/GVL_iXlinker.EtherCAT_Master_EQxxxx.Beckhoff_EQ3xxx.Beckhoff_EQ3xxxEK1122.A_0013_EQ3314_0002_0021.TC_TCInputs_Channel_1.Status/TxPDO_State <-> TC TCInputs Channel 1/Status/TxPDO State
//     PlcTask Inputs/GVL_iXlinker.EtherCAT_Master_EQxxxx.Beckhoff_EQ3xxx.Beckhoff_EQ3xxxEK1122.A_0013_EQ3314_0002_0021.TC_TCInputs_Channel_2.Status/TxPDO_State <-> TC TCInputs Channel 2/Status/TxPDO State
//     PlcTask Inputs/GVL_iXlinker.EtherCAT_Master_EQxxxx.Beckhoff_EQ3xxx.Beckhoff_EQ3xxxEK1122.A_0013_EQ3314_0002_0021.TC_TCInputs_Channel_3.Status/TxPDO_State <-> TC TCInputs Channel 3/Status/TxPDO State
//     PlcTask Inputs/GVL_iXlinker.EtherCAT_Master_EQxxxx.Beckhoff_EQ3xxx.Beckhoff_EQ3xxxEK1122.A_0013_EQ3314_0002_0021.TC_TCInputs_Channel_4.Status/TxPDO_State <-> TC TCInputs Channel 4/Status/TxPDO State
//     PlcTask Inputs/GVL_iXlinker.EtherCAT_Master_EQxxxx.Beckhoff_EQ3xxx.Beckhoff_EQ3xxxEK1122.A_0013_EQ3314_0002_0021.TC_TCInputs_Channel_1.Status/TxPDO_Toggle <-> TC TCInputs Channel 1/Status/TxPDO Toggle
//     PlcTask Inputs/GVL_iXlinker.EtherCAT_Master_EQxxxx.Beckhoff_EQ3xxx.Beckhoff_EQ3xxxEK1122.A_0013_EQ3314_0002_0021.TC_TCInputs_Channel_2.Status/TxPDO_Toggle <-> TC TCInputs Channel 2/Status/TxPDO Toggle
//     PlcTask Inputs/GVL_iXlinker.EtherCAT_Master_EQxxxx.Beckhoff_EQ3xxx.Beckhoff_EQ3xxxEK1122.A_0013_EQ3314_0002_0021.TC_TCInputs_Channel_3.Status/TxPDO_Toggle <-> TC TCInputs Channel 3/Status/TxPDO Toggle
//     PlcTask Inputs/GVL_iXlinker.EtherCAT_Master_EQxxxx.Beckhoff_EQ3xxx.Beckhoff_EQ3xxxEK1122.A_0013_EQ3314_0002_0021.TC_TCInputs_Channel_4.Status/TxPDO_Toggle <-> TC TCInputs Channel 4/Status/TxPDO Toggle
//     PlcTask Inputs/GVL_iXlinker.EtherCAT_Master_EQxxxx.Beckhoff_EQ3xxx.Beckhoff_EQ3xxxEK1122.A_0013_EQ3314_0002_0021.TC_TCInputs_Channel_1.Value <-> TC TCInputs Channel 1/Value
//     PlcTask Inputs/GVL_iXlinker.EtherCAT_Master_EQxxxx.Beckhoff_EQ3xxx.Beckhoff_EQ3xxxEK1122.A_0013_EQ3314_0002_0021.TC_TCInputs_Channel_2.Value <-> TC TCInputs Channel 2/Value
//     PlcTask Inputs/GVL_iXlinker.EtherCAT_Master_EQxxxx.Beckhoff_EQ3xxx.Beckhoff_EQ3xxxEK1122.A_0013_EQ3314_0002_0021.TC_TCInputs_Channel_3.Value <-> TC TCInputs Channel 3/Value
//     PlcTask Inputs/GVL_iXlinker.EtherCAT_Master_EQxxxx.Beckhoff_EQ3xxx.Beckhoff_EQ3xxxEK1122.A_0013_EQ3314_0002_0021.TC_TCInputs_Channel_4.Value <-> TC TCInputs Channel 4/Value
//     PlcTask Inputs/GVL_iXlinker.EtherCAT_Master_EQxxxx.Beckhoff_EQ3xxx.Beckhoff_EQ3xxxEK1122.A_0013_EQ3314_0002_0021.WcState.WcState <-> WcState/WcState
//     PlcTask Inputs/GVL_iXlinker.EtherCAT_Master_EQxxxx.Beckhoff_EQ3xxx.Beckhoff_EQ3xxxEK1122.A_0013_EQ3314_0002_0021.WcState.InputToggle <-> WcState/InputToggle
//     PlcTask Inputs/GVL_iXlinker.EtherCAT_Master_EQxxxx.Beckhoff_EQ3xxx.Beckhoff_EQ3xxxEK1122.A_0013_EQ3314_0002_0021.InfoData.AdsAddr <-> InfoData/AdsAddr
//     PlcTask Inputs/GVL_iXlinker.EtherCAT_Master_EQxxxx.Beckhoff_EQ3xxx.Beckhoff_EQ3xxxEK1122.A_0013_EQ3314_0002_0021.InfoData.State <-> InfoData/State
//   PLC/PLC Instance <-> EtherCAT Master EQxxxx/Beckhoff EQ3xxx/Beckhoff EQ3xxxEK1122/A_0014(EQ3314-0002-0022)
//     PlcTask Inputs/GVL_iXlinker.EtherCAT_Master_EQxxxx.Beckhoff_EQ3xxx.Beckhoff_EQ3xxxEK1122.A_0014_EQ3314_0002_0022.TC_Inputs_Channel_1.Status/Underrange <-> TC Inputs Channel 1/Status/Underrange
//     PlcTask Inputs/GVL_iXlinker.EtherCAT_Master_EQxxxx.Beckhoff_EQ3xxx.Beckhoff_EQ3xxxEK1122.A_0014_EQ3314_0002_0022.TC_Inputs_Channel_2.Status/Underrange <-> TC Inputs Channel 2/Status/Underrange
//     PlcTask Inputs/GVL_iXlinker.EtherCAT_Master_EQxxxx.Beckhoff_EQ3xxx.Beckhoff_EQ3xxxEK1122.A_0014_EQ3314_0002_0022.TC_Inputs_Channel_3.Status/Underrange <-> TC Inputs Channel 3/Status/Underrange
//     PlcTask Inputs/GVL_iXlinker.EtherCAT_Master_EQxxxx.Beckhoff_EQ3xxx.Beckhoff_EQ3xxxEK1122.A_0014_EQ3314_0002_0022.TC_Inputs_Channel_4.Status/Underrange <-> TC Inputs Channel 4/Status/Underrange
//     PlcTask Inputs/GVL_iXlinker.EtherCAT_Master_EQxxxx.Beckhoff_EQ3xxx.Beckhoff_EQ3xxxEK1122.A_0014_EQ3314_0002_0022.TC_Inputs_Channel_1.Status/Overrange <-> TC Inputs Channel 1/Status/Overrange
//     PlcTask Inputs/GVL_iXlinker.EtherCAT_Master_EQxxxx.Beckhoff_EQ3xxx.Beckhoff_EQ3xxxEK1122.A_0014_EQ3314_0002_0022.TC_Inputs_Channel_2.Status/Overrange <-> TC Inputs Channel 2/Status/Overrange
//     PlcTask Inputs/GVL_iXlinker.EtherCAT_Master_EQxxxx.Beckhoff_EQ3xxx.Beckhoff_EQ3xxxEK1122.A_0014_EQ3314_0002_0022.TC_Inputs_Channel_3.Status/Overrange <-> TC Inputs Channel 3/Status/Overrange
//     PlcTask Inputs/GVL_iXlinker.EtherCAT_Master_EQxxxx.Beckhoff_EQ3xxx.Beckhoff_EQ3xxxEK1122.A_0014_EQ3314_0002_0022.TC_Inputs_Channel_4.Status/Overrange <-> TC Inputs Channel 4/Status/Overrange
//     PlcTask Inputs/GVL_iXlinker.EtherCAT_Master_EQxxxx.Beckhoff_EQ3xxx.Beckhoff_EQ3xxxEK1122.A_0014_EQ3314_0002_0022.TC_Inputs_Channel_1.Status/Limit_1 <-> TC Inputs Channel 1/Status/Limit 1
//     PlcTask Inputs/GVL_iXlinker.EtherCAT_Master_EQxxxx.Beckhoff_EQ3xxx.Beckhoff_EQ3xxxEK1122.A_0014_EQ3314_0002_0022.TC_Inputs_Channel_1.Status/Limit_2 <-> TC Inputs Channel 1/Status/Limit 2
//     PlcTask Inputs/GVL_iXlinker.EtherCAT_Master_EQxxxx.Beckhoff_EQ3xxx.Beckhoff_EQ3xxxEK1122.A_0014_EQ3314_0002_0022.TC_Inputs_Channel_2.Status/Limit_1 <-> TC Inputs Channel 2/Status/Limit 1
//     PlcTask Inputs/GVL_iXlinker.EtherCAT_Master_EQxxxx.Beckhoff_EQ3xxx.Beckhoff_EQ3xxxEK1122.A_0014_EQ3314_0002_0022.TC_Inputs_Channel_2.Status/Limit_2 <-> TC Inputs Channel 2/Status/Limit 2
//     PlcTask Inputs/GVL_iXlinker.EtherCAT_Master_EQxxxx.Beckhoff_EQ3xxx.Beckhoff_EQ3xxxEK1122.A_0014_EQ3314_0002_0022.TC_Inputs_Channel_3.Status/Limit_1 <-> TC Inputs Channel 3/Status/Limit 1
//     PlcTask Inputs/GVL_iXlinker.EtherCAT_Master_EQxxxx.Beckhoff_EQ3xxx.Beckhoff_EQ3xxxEK1122.A_0014_EQ3314_0002_0022.TC_Inputs_Channel_3.Status/Limit_2 <-> TC Inputs Channel 3/Status/Limit 2
//     PlcTask Inputs/GVL_iXlinker.EtherCAT_Master_EQxxxx.Beckhoff_EQ3xxx.Beckhoff_EQ3xxxEK1122.A_0014_EQ3314_0002_0022.TC_Inputs_Channel_4.Status/Limit_1 <-> TC Inputs Channel 4/Status/Limit 1
//     PlcTask Inputs/GVL_iXlinker.EtherCAT_Master_EQxxxx.Beckhoff_EQ3xxx.Beckhoff_EQ3xxxEK1122.A_0014_EQ3314_0002_0022.TC_Inputs_Channel_4.Status/Limit_2 <-> TC Inputs Channel 4/Status/Limit 2
//     PlcTask Inputs/GVL_iXlinker.EtherCAT_Master_EQxxxx.Beckhoff_EQ3xxx.Beckhoff_EQ3xxxEK1122.A_0014_EQ3314_0002_0022.TC_Inputs_Channel_1.Status/Error <-> TC Inputs Channel 1/Status/Error
//     PlcTask Inputs/GVL_iXlinker.EtherCAT_Master_EQxxxx.Beckhoff_EQ3xxx.Beckhoff_EQ3xxxEK1122.A_0014_EQ3314_0002_0022.TC_Inputs_Channel_2.Status/Error <-> TC Inputs Channel 2/Status/Error
//     PlcTask Inputs/GVL_iXlinker.EtherCAT_Master_EQxxxx.Beckhoff_EQ3xxx.Beckhoff_EQ3xxxEK1122.A_0014_EQ3314_0002_0022.TC_Inputs_Channel_3.Status/Error <-> TC Inputs Channel 3/Status/Error
//     PlcTask Inputs/GVL_iXlinker.EtherCAT_Master_EQxxxx.Beckhoff_EQ3xxx.Beckhoff_EQ3xxxEK1122.A_0014_EQ3314_0002_0022.TC_Inputs_Channel_4.Status/Error <-> TC Inputs Channel 4/Status/Error
//     PlcTask Inputs/GVL_iXlinker.EtherCAT_Master_EQxxxx.Beckhoff_EQ3xxx.Beckhoff_EQ3xxxEK1122.A_0014_EQ3314_0002_0022.TC_Inputs_Channel_1.Status/TxPDO_State <-> TC Inputs Channel 1/Status/TxPDO State
//     PlcTask Inputs/GVL_iXlinker.EtherCAT_Master_EQxxxx.Beckhoff_EQ3xxx.Beckhoff_EQ3xxxEK1122.A_0014_EQ3314_0002_0022.TC_Inputs_Channel_2.Status/TxPDO_State <-> TC Inputs Channel 2/Status/TxPDO State
//     PlcTask Inputs/GVL_iXlinker.EtherCAT_Master_EQxxxx.Beckhoff_EQ3xxx.Beckhoff_EQ3xxxEK1122.A_0014_EQ3314_0002_0022.TC_Inputs_Channel_3.Status/TxPDO_State <-> TC Inputs Channel 3/Status/TxPDO State
//     PlcTask Inputs/GVL_iXlinker.EtherCAT_Master_EQxxxx.Beckhoff_EQ3xxx.Beckhoff_EQ3xxxEK1122.A_0014_EQ3314_0002_0022.TC_Inputs_Channel_4.Status/TxPDO_State <-> TC Inputs Channel 4/Status/TxPDO State
//     PlcTask Inputs/GVL_iXlinker.EtherCAT_Master_EQxxxx.Beckhoff_EQ3xxx.Beckhoff_EQ3xxxEK1122.A_0014_EQ3314_0002_0022.TC_Inputs_Channel_1.Status/TxPDO_Toggle <-> TC Inputs Channel 1/Status/TxPDO Toggle
//     PlcTask Inputs/GVL_iXlinker.EtherCAT_Master_EQxxxx.Beckhoff_EQ3xxx.Beckhoff_EQ3xxxEK1122.A_0014_EQ3314_0002_0022.TC_Inputs_Channel_2.Status/TxPDO_Toggle <-> TC Inputs Channel 2/Status/TxPDO Toggle
//     PlcTask Inputs/GVL_iXlinker.EtherCAT_Master_EQxxxx.Beckhoff_EQ3xxx.Beckhoff_EQ3xxxEK1122.A_0014_EQ3314_0002_0022.TC_Inputs_Channel_3.Status/TxPDO_Toggle <-> TC Inputs Channel 3/Status/TxPDO Toggle
//     PlcTask Inputs/GVL_iXlinker.EtherCAT_Master_EQxxxx.Beckhoff_EQ3xxx.Beckhoff_EQ3xxxEK1122.A_0014_EQ3314_0002_0022.TC_Inputs_Channel_4.Status/TxPDO_Toggle <-> TC Inputs Channel 4/Status/TxPDO Toggle
//     PlcTask Inputs/GVL_iXlinker.EtherCAT_Master_EQxxxx.Beckhoff_EQ3xxx.Beckhoff_EQ3xxxEK1122.A_0014_EQ3314_0002_0022.TC_Inputs_Channel_1.Value <-> TC Inputs Channel 1/Value
//     PlcTask Inputs/GVL_iXlinker.EtherCAT_Master_EQxxxx.Beckhoff_EQ3xxx.Beckhoff_EQ3xxxEK1122.A_0014_EQ3314_0002_0022.TC_Inputs_Channel_2.Value <-> TC Inputs Channel 2/Value
//     PlcTask Inputs/GVL_iXlinker.EtherCAT_Master_EQxxxx.Beckhoff_EQ3xxx.Beckhoff_EQ3xxxEK1122.A_0014_EQ3314_0002_0022.TC_Inputs_Channel_3.Value <-> TC Inputs Channel 3/Value
//     PlcTask Inputs/GVL_iXlinker.EtherCAT_Master_EQxxxx.Beckhoff_EQ3xxx.Beckhoff_EQ3xxxEK1122.A_0014_EQ3314_0002_0022.TC_Inputs_Channel_4.Value <-> TC Inputs Channel 4/Value
//     PlcTask Inputs/GVL_iXlinker.EtherCAT_Master_EQxxxx.Beckhoff_EQ3xxx.Beckhoff_EQ3xxxEK1122.A_0014_EQ3314_0002_0022.WcState.WcState <-> WcState/WcState
//     PlcTask Inputs/GVL_iXlinker.EtherCAT_Master_EQxxxx.Beckhoff_EQ3xxx.Beckhoff_EQ3xxxEK1122.A_0014_EQ3314_0002_0022.WcState.InputToggle <-> WcState/InputToggle
//     PlcTask Inputs/GVL_iXlinker.EtherCAT_Master_EQxxxx.Beckhoff_EQ3xxx.Beckhoff_EQ3xxxEK1122.A_0014_EQ3314_0002_0022.InfoData.AdsAddr <-> InfoData/AdsAddr
//     PlcTask Inputs/GVL_iXlinker.EtherCAT_Master_EQxxxx.Beckhoff_EQ3xxx.Beckhoff_EQ3xxxEK1122.A_0014_EQ3314_0002_0022.InfoData.State <-> InfoData/State
//   PLC/PLC Instance <-> EtherCAT_Master_EQxxxx
//     PlcTask Inputs/GVL_iXlinker.EtherCAT_Master_EQxxxx.SyncUnits._default._unreferenced.WcState.WcState <-> SyncUnits/<default>/<unreferenced>/WcState/WcState
//     PlcTask Inputs/GVL_iXlinker.EtherCAT_Master_EQxxxx.SyncUnits._default._unreferenced.InfoData.ObjectId <-> SyncUnits/<default>/<unreferenced>/InfoData/ObjectId
//     PlcTask Inputs/GVL_iXlinker.EtherCAT_Master_EQxxxx.SyncUnits._default._unreferenced.InfoData.State <-> SyncUnits/<default>/<unreferenced>/InfoData/State
//     PlcTask Inputs/GVL_iXlinker.EtherCAT_Master_EQxxxx.SyncUnits._default._unreferenced.InfoData.SlaveCount <-> SyncUnits/<default>/<unreferenced>/InfoData/SlaveCount
//     PlcTask Inputs/GVL_iXlinker.EtherCAT_Master_EQxxxx.SyncUnits._default.PlcTask.WcState.WcState <-> SyncUnits/<default>/PlcTask/WcState/WcState
//     PlcTask Inputs/GVL_iXlinker.EtherCAT_Master_EQxxxx.SyncUnits._default.PlcTask.InfoData.ObjectId <-> SyncUnits/<default>/PlcTask/InfoData/ObjectId
//     PlcTask Inputs/GVL_iXlinker.EtherCAT_Master_EQxxxx.SyncUnits._default.PlcTask.InfoData.State <-> SyncUnits/<default>/PlcTask/InfoData/State
//     PlcTask Inputs/GVL_iXlinker.EtherCAT_Master_EQxxxx.SyncUnits._default.PlcTask.InfoData.SlaveCount <-> SyncUnits/<default>/PlcTask/InfoData/SlaveCount
//     PlcTask Inputs/GVL_iXlinker.EtherCAT_Master_EQxxxx.Inputs.SlaveCount <-> Inputs/SlaveCount
//     PlcTask Inputs/GVL_iXlinker.EtherCAT_Master_EQxxxx.Inputs.DevState <-> Inputs/DevState
//     PlcTask Inputs/GVL_iXlinker.EtherCAT_Master_EQxxxx.Inputs.Frm{0..25}State <-> Inputs/Frm{0..25}State  (26 links)
//     PlcTask Inputs/GVL_iXlinker.EtherCAT_Master_EQxxxx.Inputs.Frm{0..25}WcState <-> Inputs/Frm{0..25}WcState  (26 links)
//     PlcTask Inputs/GVL_iXlinker.EtherCAT_Master_EQxxxx.Inputs.Frm{0..25}InputToggle <-> Inputs/Frm{0..25}InputToggle  (26 links)
//     PlcTask Outputs/GVL_iXlinker.EtherCAT_Master_EQxxxx.Outputs.DevCtrl <-> Outputs/DevCtrl
//     PlcTask Outputs/GVL_iXlinker.EtherCAT_Master_EQxxxx.Outputs.Frm{0..25}Ctrl <-> Outputs/Frm{0..25}Ctrl  (26 links)
//     PlcTask Outputs/GVL_iXlinker.EtherCAT_Master_EQxxxx.Outputs.Frm{0..25}WcCtrl <-> Outputs/Frm{0..25}WcCtrl  (26 links)
//     PlcTask Inputs/GVL_iXlinker.EtherCAT_Master_EQxxxx.InfoData.ChangeCount <-> InfoData/ChangeCount
//     PlcTask Inputs/GVL_iXlinker.EtherCAT_Master_EQxxxx.InfoData.DevId <-> InfoData/DevId
//     PlcTask Inputs/GVL_iXlinker.EtherCAT_Master_EQxxxx.InfoData.AmsNetId <-> InfoData/AmsNetId
//     PlcTask Inputs/GVL_iXlinker.EtherCAT_Master_EQxxxx.InfoData.CfgSlaveCount <-> InfoData/CfgSlaveCount
//     PlcTask Inputs/GVL_iXlinker.EtherCAT_Master_EQxxxx.InfoData.DcToTcTimeOffset <-> InfoData/DcToTcTimeOffset
//     PlcTask Inputs/GVL_iXlinker.EtherCAT_Master_EQxxxx.InfoData.DcToExtTimeOffset <-> InfoData/DcToExtTimeOffset

CONFIGURATION PLC
    RESOURCE PLC ON TwinCAT3
        TASK PlcTask(INTERVAL := T#10ms, PRIORITY := 20);
        PROGRAM MAIN WITH PlcTask : MAIN;
    END_RESOURCE
END_CONFIGURATION

// ---- DUTs/IO/PdoEntries/Status_B0753356.TcDUT
{attribute 'GeneratedUsingTerminal: EQ3174-0002-0016'}
{attribute addProperty BoxType "EQ3174-0002-0016"}
{attribute addProperty Id "UnderrangeBOOL1OverrangeBOOL1Limit_1BYTE1Limit_2BYTE1ErrorBOOL1Sync_errorBOOL1TxPDO_StateBOOL1TxPDO_ToggleBOOL1"}
{attribute addProperty CRC "2960470870"}
{attribute addProperty Size "8"}
TYPE Status_B0753356 :
STRUCT
	{attribute addProperty Name "Underrange"}
	Underrange : BOOL;
	{attribute addProperty Name "Overrange"}
	Overrange : BOOL;
	{attribute addProperty Name "Limit_1"}
	Limit_1 : BYTE;
	{attribute addProperty Name "Limit_2"}
	Limit_2 : BYTE;
	{attribute addProperty Name "Error"}
	Error : BOOL;
	{attribute addProperty Name "Sync_error"}
	Sync_error : BOOL;
	{attribute addProperty Name "TxPDO_State"}
	TxPDO_State : BOOL;
	{attribute addProperty Name "TxPDO_Toggle"}
	TxPDO_Toggle : BOOL;
END_STRUCT
END_TYPE

// ---- DUTs/IO/PdoEntries/Status_F2CE6D91.TcDUT
{attribute 'GeneratedUsingTerminal: EQ3204-0002-0021'}
{attribute addProperty BoxType "EQ3204-0002-0021"}
{attribute addProperty Id "UnderrangeBOOL1OverrangeBOOL1Limit_1BYTE1Limit_2BYTE1ErrorBOOL1TxPDO_StateBOOL1TxPDO_ToggleBOOL1"}
{attribute addProperty CRC "4073614737"}
{attribute addProperty Size "7"}
TYPE Status_F2CE6D91 :
STRUCT
	{attribute addProperty Name "Underrange"}
	Underrange : BOOL;
	{attribute addProperty Name "Overrange"}
	Overrange : BOOL;
	{attribute addProperty Name "Limit_1"}
	Limit_1 : BYTE;
	{attribute addProperty Name "Limit_2"}
	Limit_2 : BYTE;
	{attribute addProperty Name "Error"}
	Error : BOOL;
	{attribute addProperty Name "TxPDO_State"}
	TxPDO_State : BOOL;
	{attribute addProperty Name "TxPDO_Toggle"}
	TxPDO_Toggle : BOOL;
END_STRUCT
END_TYPE

// ---- DUTs/IO/PDOs/InfoData_6F19DB2B.TcDUT
{attribute 'GeneratedUsingTerminal: EK1100-0000-0018'}
{attribute addProperty BoxType "EK1100-0000-0018"}
{attribute addProperty Id "StateAT %I*UINT2"}
{attribute addProperty CRC "1863965483"}
{attribute addProperty Size "2"}
TYPE InfoData_6F19DB2B :
STRUCT
	{attribute addProperty Name "State"}
	State AT %I* : UINT;
END_STRUCT
END_TYPE

// ---- DUTs/IO/PDOs/Channel_830843C1.TcDUT
{attribute 'GeneratedUsingTerminal: EQ1008-0002-0016'}
{attribute addProperty BoxType "EQ1008-0002-0016"}
{attribute addProperty Id "InputAT %I*BOOL1"}
{attribute addProperty CRC "2198356929"}
{attribute addProperty Size "1"}
TYPE Channel_830843C1 EXTENDS InputBase_8311D824 :
STRUCT
	{attribute addProperty Name "Input"}
	Input AT %I* : BOOL;
END_STRUCT
END_TYPE

// ---- DUTs/IO/PDOs/WcState_9091E0EB.TcDUT
{attribute 'GeneratedUsingTerminal: EQ1008-0002-0016'}
{attribute addProperty BoxType "EQ1008-0002-0016"}
{attribute addProperty Id "WcStateAT %I*BOOL1InputToggleAT %I*BOOL1"}
{attribute addProperty CRC "2425479403"}
{attribute addProperty Size "2"}
TYPE WcState_9091E0EB :
STRUCT
	{attribute addProperty Name "WcState"}
	WcState AT %I* : BOOL;
	{attribute addProperty Name "InputToggle"}
	InputToggle AT %I* : BOOL;
END_STRUCT
END_TYPE

// ---- DUTs/IO/PDOs/Channel_42CA91F7.TcDUT
{attribute 'GeneratedUsingTerminal: EQ2008-0002-0016'}
{attribute addProperty BoxType "EQ2008-0002-0016"}
{attribute addProperty Id "OutputAT %Q*BOOL1"}
{attribute addProperty CRC "1120571895"}
{attribute addProperty Size "1"}
TYPE Channel_42CA91F7 EXTENDS OutputBase_10CEE7DE :
STRUCT
	{attribute addProperty Name "Output"}
	Output AT %Q* : BOOL;
END_STRUCT
END_TYPE

// ---- DUTs/IO/PDOs/WcState_0B2B16F9.TcDUT
{attribute 'GeneratedUsingTerminal: EQ2008-0002-0016'}
{attribute addProperty BoxType "EQ2008-0002-0016"}
{attribute addProperty Id "WcStateAT %I*BOOL1"}
{attribute addProperty CRC "187373305"}
{attribute addProperty Size "1"}
TYPE WcState_0B2B16F9 :
STRUCT
	{attribute addProperty Name "WcState"}
	WcState AT %I* : BOOL;
END_STRUCT
END_TYPE

// ---- DUTs/IO/PDOs/AI_Standard_Channel_A8DF64E3.TcDUT
{attribute 'GeneratedUsingTerminal: EQ3174-0002-0016'}
{attribute addProperty BoxType "EQ3174-0002-0016"}
{attribute addProperty Id "StatusAT %I*Status_B07533568ValueAT %I*INT2"}
{attribute addProperty CRC "2833212643"}
{attribute addProperty Size "10"}
TYPE AI_Standard_Channel_A8DF64E3 EXTENDS InputBase_8311D824 :
STRUCT
	{attribute addProperty Name "Status"}
	Status AT %I* : Status_B0753356;
	{attribute addProperty Name "Value"}
	Value AT %I* : INT;
END_STRUCT
END_TYPE

// ---- DUTs/IO/PDOs/InfoData_32EB74EA.TcDUT
{attribute 'GeneratedUsingTerminal: EQ3174-0002-0016'}
{attribute addProperty BoxType "EQ3174-0002-0016"}
{attribute addProperty Id "AdsAddrAT %I*AMSADDR8StateAT %I*UINT2"}
{attribute addProperty CRC "854291690"}
{attribute addProperty Size "10"}
TYPE InfoData_32EB74EA EXTENDS InputBase_8311D824 :
STRUCT
	{attribute addProperty Name "AdsAddr"}
	AdsAddr AT %I* : AMSADDR;
	{attribute addProperty Name "State"}
	State AT %I* : UINT;
END_STRUCT
END_TYPE

// ---- DUTs/IO/PDOs/RTD_RTDInputs_Channel_A8DF64E3.TcDUT
{attribute 'GeneratedUsingTerminal: EQ3204-0002-0016'}
{attribute addProperty BoxType "EQ3204-0002-0016"}
{attribute addProperty Id "StatusAT %I*Status_B07533568ValueAT %I*INT2"}
{attribute addProperty CRC "2833212643"}
{attribute addProperty Size "10"}
TYPE RTD_RTDInputs_Channel_A8DF64E3 EXTENDS InputBase_8311D824 :
STRUCT
	{attribute addProperty Name "Status"}
	Status AT %I* : Status_B0753356;
	{attribute addProperty Name "Value"}
	Value AT %I* : INT;
END_STRUCT
END_TYPE

// ---- DUTs/IO/PDOs/AI_Standard_Channel_4A394481.TcDUT
{attribute 'GeneratedUsingTerminal: EQ3204-0002-0021'}
{attribute addProperty BoxType "EQ3204-0002-0021"}
{attribute addProperty Id "StatusAT %I*Status_F2CE6D917ValueAT %I*INT2"}
{attribute addProperty CRC "1245267073"}
{attribute addProperty Size "9"}
TYPE AI_Standard_Channel_4A394481 EXTENDS InputBase_8311D824 :
STRUCT
	{attribute addProperty Name "Status"}
	Status AT %I* : Status_F2CE6D91;
	{attribute addProperty Name "Value"}
	Value AT %I* : INT;
END_STRUCT
END_TYPE

// ---- DUTs/IO/PDOs/TC_TCInputs_Channel_A8DF64E3.TcDUT
{attribute 'GeneratedUsingTerminal: EQ3314-0002-0016'}
{attribute addProperty BoxType "EQ3314-0002-0016"}
{attribute addProperty Id "StatusAT %I*Status_B07533568ValueAT %I*INT2"}
{attribute addProperty CRC "2833212643"}
{attribute addProperty Size "10"}
TYPE TC_TCInputs_Channel_A8DF64E3 EXTENDS InputBase_8311D824 :
STRUCT
	{attribute addProperty Name "Status"}
	Status AT %I* : Status_B0753356;
	{attribute addProperty Name "Value"}
	Value AT %I* : INT;
END_STRUCT
END_TYPE

// ---- DUTs/IO/PDOs/InfoData_E68C61CD.TcDUT
{attribute 'GeneratedUsingTerminal: IODEVICETYPE_ETHERCATPROT'}
{attribute addProperty BoxType "IODEVICETYPE_ETHERCATPROT"}
{attribute addProperty Id "ChangeCountAT %I*UINT2DevIdAT %I*UINT2AmsNetIdAT %I*AMSNETID6CfgSlaveCountAT %I*UINT2DcToTcTimeOffsetAT %I*LINT8DcToExtTimeOffsetAT %I*LINT8"}
{attribute addProperty CRC "3867959757"}
{attribute addProperty Size "28"}
TYPE InfoData_E68C61CD EXTENDS InputBase_8311D824 :
STRUCT
	{attribute addProperty Name "ChangeCount"}
	ChangeCount AT %I* : UINT;
	{attribute addProperty Name "DevId"}
	DevId AT %I* : UINT;
	{attribute addProperty Name "AmsNetId"}
	AmsNetId AT %I* : AMSNETID;
	{attribute addProperty Name "CfgSlaveCount"}
	CfgSlaveCount AT %I* : UINT;
	{attribute addProperty Name "DcToTcTimeOffset"}
	DcToTcTimeOffset AT %I* : LINT;
	{attribute addProperty Name "DcToExtTimeOffset"}
	DcToExtTimeOffset AT %I* : LINT;
END_STRUCT
END_TYPE

// ---- DUTs/IO/PDOs/InfoData_2A97D6CF.TcDUT
{attribute 'GeneratedUsingTerminal: IODEVICETYPE_ETHERCATPROT'}
{attribute addProperty BoxType "IODEVICETYPE_ETHERCATPROT"}
{attribute addProperty Id "ObjectIdAT %I*OTCID4StateAT %I*UINT2SlaveCountAT %I*UINT2"}
{attribute addProperty CRC "714593999"}
{attribute addProperty Size "8"}
TYPE InfoData_2A97D6CF EXTENDS InputBase_8311D824 :
STRUCT
	{attribute addProperty Name "ObjectId"}
	ObjectId AT %I* : OTCID;
	{attribute addProperty Name "State"}
	State AT %I* : UINT;
	{attribute addProperty Name "SlaveCount"}
	SlaveCount AT %I* : UINT;
END_STRUCT
END_TYPE

// ---- DUTs/IO/PDOs/Inputs_25A0042B.TcDUT
{attribute 'GeneratedUsingTerminal: IODEVICETYPE_ETHERCATPROT'}
{attribute addProperty BoxType "IODEVICETYPE_ETHERCATPROT"}
{attribute addProperty Id "SlaveCountAT %I*UINT2DevStateAT %I*UINT2Frm0StateAT %I*UINT2Frm0WcStateAT %I*UINT2Frm0InputToggleAT %I*UINT2Frm1StateAT %I*UINT2Frm1WcStateAT %I*UINT2Frm1InputToggleAT %I*UINT2Frm2StateAT %I*UINT2Frm2WcStateAT %I*UINT2Frm2InputToggleAT %I*UINT2Frm3StateAT %I*UINT2Frm3WcStateAT %I*UINT2Frm3InputToggleAT %I*UINT2Frm4StateAT %I*UINT2Frm4WcStateAT %I*UINT2Frm4InputToggleAT %I*UINT2Frm5StateAT %I*UINT2Frm5WcStateAT %I*UINT2Frm5InputToggleAT %I*UINT2Frm6StateAT %I*UINT2Frm6WcStateAT %I*UINT2Frm6InputToggleAT %I*UINT2Frm7StateAT %I*UINT2Frm7WcStateAT %I*UINT2Frm7InputToggleAT %I*UINT2Frm8StateAT %I*UINT2Frm8WcStateAT %I*UINT2Frm8InputToggleAT %I*UINT2Frm9StateAT %I*UINT2Frm9WcStateAT %I*UINT2Frm9InputToggleAT %I*UINT2Frm10StateAT %I*UINT2Frm10WcStateAT %I*UINT2Frm10InputToggleAT %I*UINT2Frm11StateAT %I*UINT2Frm11WcStateAT %I*UINT2Frm11InputToggleAT %I*UINT2Frm12StateAT %I*UINT2Frm12WcStateAT %I*UINT2Frm12InputToggleAT %I*UINT2Frm13StateAT %I*UINT2Frm13WcStateAT %I*UINT2Frm13InputToggleAT %I*UINT2Frm14StateAT %I*UINT2Frm14WcStateAT %I*UINT2Frm14InputToggleAT %I*UINT2Frm15StateAT %I*UINT2Frm15WcStateAT %I*UINT2Frm15InputToggleAT %I*UINT2Frm16StateAT %I*UINT2Frm16WcStateAT %I*UINT2Frm16InputToggleAT %I*UINT2Frm17StateAT %I*UINT2Frm17WcStateAT %I*UINT2Frm17InputToggleAT %I*UINT2Frm18StateAT %I*UINT2Frm18WcStateAT %I*UINT2Frm18InputToggleAT %I*UINT2Frm19StateAT %I*UINT2Frm19WcStateAT %I*UINT2Frm19InputToggleAT %I*UINT2Frm20StateAT %I*UINT2Frm20WcStateAT %I*UINT2Frm20InputToggleAT %I*UINT2Frm21StateAT %I*UINT2Frm21WcStateAT %I*UINT2Frm21InputToggleAT %I*UINT2Frm22StateAT %I*UINT2Frm22WcStateAT %I*UINT2Frm22InputToggleAT %I*UINT2Frm23StateAT %I*UINT2Frm23WcStateAT %I*UINT2Frm23InputToggleAT %I*UINT2Frm24StateAT %I*UINT2Frm24WcStateAT %I*UINT2Frm24InputToggleAT %I*UINT2Frm25StateAT %I*UINT2Frm25WcStateAT %I*UINT2Frm25InputToggleAT %I*UINT2"}
{attribute addProperty CRC "631243819"}
{attribute addProperty Size "160"}
TYPE Inputs_25A0042B EXTENDS InputBase_8311D824 :
STRUCT
	{attribute addProperty Name "SlaveCount"}
	SlaveCount AT %I* : UINT;
	{attribute addProperty Name "DevState"}
	DevState AT %I* : UINT;
	{attribute addProperty Name "Frm0State"}
	Frm0State AT %I* : UINT;
	{attribute addProperty Name "Frm0WcState"}
	Frm0WcState AT %I* : UINT;
	{attribute addProperty Name "Frm0InputToggle"}
	Frm0InputToggle AT %I* : UINT;
	{attribute addProperty Name "Frm1State"}
	Frm1State AT %I* : UINT;
	{attribute addProperty Name "Frm1WcState"}
	Frm1WcState AT %I* : UINT;
	{attribute addProperty Name "Frm1InputToggle"}
	Frm1InputToggle AT %I* : UINT;
	{attribute addProperty Name "Frm2State"}
	Frm2State AT %I* : UINT;
	{attribute addProperty Name "Frm2WcState"}
	Frm2WcState AT %I* : UINT;
	{attribute addProperty Name "Frm2InputToggle"}
	Frm2InputToggle AT %I* : UINT;
	{attribute addProperty Name "Frm3State"}
	Frm3State AT %I* : UINT;
	{attribute addProperty Name "Frm3WcState"}
	Frm3WcState AT %I* : UINT;
	{attribute addProperty Name "Frm3InputToggle"}
	Frm3InputToggle AT %I* : UINT;
	{attribute addProperty Name "Frm4State"}
	Frm4State AT %I* : UINT;
	{attribute addProperty Name "Frm4WcState"}
	Frm4WcState AT %I* : UINT;
	{attribute addProperty Name "Frm4InputToggle"}
	Frm4InputToggle AT %I* : UINT;
	{attribute addProperty Name "Frm5State"}
	Frm5State AT %I* : UINT;
	{attribute addProperty Name "Frm5WcState"}
	Frm5WcState AT %I* : UINT;
	{attribute addProperty Name "Frm5InputToggle"}
	Frm5InputToggle AT %I* : UINT;
	{attribute addProperty Name "Frm6State"}
	Frm6State AT %I* : UINT;
	{attribute addProperty Name "Frm6WcState"}
	Frm6WcState AT %I* : UINT;
	{attribute addProperty Name "Frm6InputToggle"}
	Frm6InputToggle AT %I* : UINT;
	{attribute addProperty Name "Frm7State"}
	Frm7State AT %I* : UINT;
	{attribute addProperty Name "Frm7WcState"}
	Frm7WcState AT %I* : UINT;
	{attribute addProperty Name "Frm7InputToggle"}
	Frm7InputToggle AT %I* : UINT;
	{attribute addProperty Name "Frm8State"}
	Frm8State AT %I* : UINT;
	{attribute addProperty Name "Frm8WcState"}
	Frm8WcState AT %I* : UINT;
	{attribute addProperty Name "Frm8InputToggle"}
	Frm8InputToggle AT %I* : UINT;
	{attribute addProperty Name "Frm9State"}
	Frm9State AT %I* : UINT;
	{attribute addProperty Name "Frm9WcState"}
	Frm9WcState AT %I* : UINT;
	{attribute addProperty Name "Frm9InputToggle"}
	Frm9InputToggle AT %I* : UINT;
	{attribute addProperty Name "Frm10State"}
	Frm10State AT %I* : UINT;
	{attribute addProperty Name "Frm10WcState"}
	Frm10WcState AT %I* : UINT;
	{attribute addProperty Name "Frm10InputToggle"}
	Frm10InputToggle AT %I* : UINT;
	{attribute addProperty Name "Frm11State"}
	Frm11State AT %I* : UINT;
	{attribute addProperty Name "Frm11WcState"}
	Frm11WcState AT %I* : UINT;
	{attribute addProperty Name "Frm11InputToggle"}
	Frm11InputToggle AT %I* : UINT;
	{attribute addProperty Name "Frm12State"}
	Frm12State AT %I* : UINT;
	{attribute addProperty Name "Frm12WcState"}
	Frm12WcState AT %I* : UINT;
	{attribute addProperty Name "Frm12InputToggle"}
	Frm12InputToggle AT %I* : UINT;
	{attribute addProperty Name "Frm13State"}
	Frm13State AT %I* : UINT;
	{attribute addProperty Name "Frm13WcState"}
	Frm13WcState AT %I* : UINT;
	{attribute addProperty Name "Frm13InputToggle"}
	Frm13InputToggle AT %I* : UINT;
	{attribute addProperty Name "Frm14State"}
	Frm14State AT %I* : UINT;
	{attribute addProperty Name "Frm14WcState"}
	Frm14WcState AT %I* : UINT;
	{attribute addProperty Name "Frm14InputToggle"}
	Frm14InputToggle AT %I* : UINT;
	{attribute addProperty Name "Frm15State"}
	Frm15State AT %I* : UINT;
	{attribute addProperty Name "Frm15WcState"}
	Frm15WcState AT %I* : UINT;
	{attribute addProperty Name "Frm15InputToggle"}
	Frm15InputToggle AT %I* : UINT;
	{attribute addProperty Name "Frm16State"}
	Frm16State AT %I* : UINT;
	{attribute addProperty Name "Frm16WcState"}
	Frm16WcState AT %I* : UINT;
	{attribute addProperty Name "Frm16InputToggle"}
	Frm16InputToggle AT %I* : UINT;
	{attribute addProperty Name "Frm17State"}
	Frm17State AT %I* : UINT;
	{attribute addProperty Name "Frm17WcState"}
	Frm17WcState AT %I* : UINT;
	{attribute addProperty Name "Frm17InputToggle"}
	Frm17InputToggle AT %I* : UINT;
	{attribute addProperty Name "Frm18State"}
	Frm18State AT %I* : UINT;
	{attribute addProperty Name "Frm18WcState"}
	Frm18WcState AT %I* : UINT;
	{attribute addProperty Name "Frm18InputToggle"}
	Frm18InputToggle AT %I* : UINT;
	{attribute addProperty Name "Frm19State"}
	Frm19State AT %I* : UINT;
	{attribute addProperty Name "Frm19WcState"}
	Frm19WcState AT %I* : UINT;
	{attribute addProperty Name "Frm19InputToggle"}
	Frm19InputToggle AT %I* : UINT;
	{attribute addProperty Name "Frm20State"}
	Frm20State AT %I* : UINT;
	{attribute addProperty Name "Frm20WcState"}
	Frm20WcState AT %I* : UINT;
	{attribute addProperty Name "Frm20InputToggle"}
	Frm20InputToggle AT %I* : UINT;
	{attribute addProperty Name "Frm21State"}
	Frm21State AT %I* : UINT;
	{attribute addProperty Name "Frm21WcState"}
	Frm21WcState AT %I* : UINT;
	{attribute addProperty Name "Frm21InputToggle"}
	Frm21InputToggle AT %I* : UINT;
	{attribute addProperty Name "Frm22State"}
	Frm22State AT %I* : UINT;
	{attribute addProperty Name "Frm22WcState"}
	Frm22WcState AT %I* : UINT;
	{attribute addProperty Name "Frm22InputToggle"}
	Frm22InputToggle AT %I* : UINT;
	{attribute addProperty Name "Frm23State"}
	Frm23State AT %I* : UINT;
	{attribute addProperty Name "Frm23WcState"}
	Frm23WcState AT %I* : UINT;
	{attribute addProperty Name "Frm23InputToggle"}
	Frm23InputToggle AT %I* : UINT;
	{attribute addProperty Name "Frm24State"}
	Frm24State AT %I* : UINT;
	{attribute addProperty Name "Frm24WcState"}
	Frm24WcState AT %I* : UINT;
	{attribute addProperty Name "Frm24InputToggle"}
	Frm24InputToggle AT %I* : UINT;
	{attribute addProperty Name "Frm25State"}
	Frm25State AT %I* : UINT;
	{attribute addProperty Name "Frm25WcState"}
	Frm25WcState AT %I* : UINT;
	{attribute addProperty Name "Frm25InputToggle"}
	Frm25InputToggle AT %I* : UINT;
END_STRUCT
END_TYPE

// ---- DUTs/IO/PDOs/Outputs_2397A10E.TcDUT
{attribute 'GeneratedUsingTerminal: IODEVICETYPE_ETHERCATPROT'}
{attribute addProperty BoxType "IODEVICETYPE_ETHERCATPROT"}
{attribute addProperty Id "DevCtrlAT %Q*UINT2Frm0CtrlAT %Q*UINT2Frm0WcCtrlAT %Q*UINT2Frm1CtrlAT %Q*UINT2Frm1WcCtrlAT %Q*UINT2Frm2CtrlAT %Q*UINT2Frm2WcCtrlAT %Q*UINT2Frm3CtrlAT %Q*UINT2Frm3WcCtrlAT %Q*UINT2Frm4CtrlAT %Q*UINT2Frm4WcCtrlAT %Q*UINT2Frm5CtrlAT %Q*UINT2Frm5WcCtrlAT %Q*UINT2Frm6CtrlAT %Q*UINT2Frm6WcCtrlAT %Q*UINT2Frm7CtrlAT %Q*UINT2Frm7WcCtrlAT %Q*UINT2Frm8CtrlAT %Q*UINT2Frm8WcCtrlAT %Q*UINT2Frm9CtrlAT %Q*UINT2Frm9WcCtrlAT %Q*UINT2Frm10CtrlAT %Q*UINT2Frm10WcCtrlAT %Q*UINT2Frm11CtrlAT %Q*UINT2Frm11WcCtrlAT %Q*UINT2Frm12CtrlAT %Q*UINT2Frm12WcCtrlAT %Q*UINT2Frm13CtrlAT %Q*UINT2Frm13WcCtrlAT %Q*UINT2Frm14CtrlAT %Q*UINT2Frm14WcCtrlAT %Q*UINT2Frm15CtrlAT %Q*UINT2Frm15WcCtrlAT %Q*UINT2Frm16CtrlAT %Q*UINT2Frm16WcCtrlAT %Q*UINT2Frm17CtrlAT %Q*UINT2Frm17WcCtrlAT %Q*UINT2Frm18CtrlAT %Q*UINT2Frm18WcCtrlAT %Q*UINT2Frm19CtrlAT %Q*UINT2Frm19WcCtrlAT %Q*UINT2Frm20CtrlAT %Q*UINT2Frm20WcCtrlAT %Q*UINT2Frm21CtrlAT %Q*UINT2Frm21WcCtrlAT %Q*UINT2Frm22CtrlAT %Q*UINT2Frm22WcCtrlAT %Q*UINT2Frm23CtrlAT %Q*UINT2Frm23WcCtrlAT %Q*UINT2Frm24CtrlAT %Q*UINT2Frm24WcCtrlAT %Q*UINT2Frm25CtrlAT %Q*UINT2Frm25WcCtrlAT %Q*UINT2"}
{attribute addProperty CRC "597139726"}
{attribute addProperty Size "106"}
TYPE Outputs_2397A10E EXTENDS OutputBase_10CEE7DE :
STRUCT
	{attribute addProperty Name "DevCtrl"}
	DevCtrl AT %Q* : UINT;
	{attribute addProperty Name "Frm0Ctrl"}
	Frm0Ctrl AT %Q* : UINT;
	{attribute addProperty Name "Frm0WcCtrl"}
	Frm0WcCtrl AT %Q* : UINT;
	{attribute addProperty Name "Frm1Ctrl"}
	Frm1Ctrl AT %Q* : UINT;
	{attribute addProperty Name "Frm1WcCtrl"}
	Frm1WcCtrl AT %Q* : UINT;
	{attribute addProperty Name "Frm2Ctrl"}
	Frm2Ctrl AT %Q* : UINT;
	{attribute addProperty Name "Frm2WcCtrl"}
	Frm2WcCtrl AT %Q* : UINT;
	{attribute addProperty Name "Frm3Ctrl"}
	Frm3Ctrl AT %Q* : UINT;
	{attribute addProperty Name "Frm3WcCtrl"}
	Frm3WcCtrl AT %Q* : UINT;
	{attribute addProperty Name "Frm4Ctrl"}
	Frm4Ctrl AT %Q* : UINT;
	{attribute addProperty Name "Frm4WcCtrl"}
	Frm4WcCtrl AT %Q* : UINT;
	{attribute addProperty Name "Frm5Ctrl"}
	Frm5Ctrl AT %Q* : UINT;
	{attribute addProperty Name "Frm5WcCtrl"}
	Frm5WcCtrl AT %Q* : UINT;
	{attribute addProperty Name "Frm6Ctrl"}
	Frm6Ctrl AT %Q* : UINT;
	{attribute addProperty Name "Frm6WcCtrl"}
	Frm6WcCtrl AT %Q* : UINT;
	{attribute addProperty Name "Frm7Ctrl"}
	Frm7Ctrl AT %Q* : UINT;
	{attribute addProperty Name "Frm7WcCtrl"}
	Frm7WcCtrl AT %Q* : UINT;
	{attribute addProperty Name "Frm8Ctrl"}
	Frm8Ctrl AT %Q* : UINT;
	{attribute addProperty Name "Frm8WcCtrl"}
	Frm8WcCtrl AT %Q* : UINT;
	{attribute addProperty Name "Frm9Ctrl"}
	Frm9Ctrl AT %Q* : UINT;
	{attribute addProperty Name "Frm9WcCtrl"}
	Frm9WcCtrl AT %Q* : UINT;
	{attribute addProperty Name "Frm10Ctrl"}
	Frm10Ctrl AT %Q* : UINT;
	{attribute addProperty Name "Frm10WcCtrl"}
	Frm10WcCtrl AT %Q* : UINT;
	{attribute addProperty Name "Frm11Ctrl"}
	Frm11Ctrl AT %Q* : UINT;
	{attribute addProperty Name "Frm11WcCtrl"}
	Frm11WcCtrl AT %Q* : UINT;
	{attribute addProperty Name "Frm12Ctrl"}
	Frm12Ctrl AT %Q* : UINT;
	{attribute addProperty Name "Frm12WcCtrl"}
	Frm12WcCtrl AT %Q* : UINT;
	{attribute addProperty Name "Frm13Ctrl"}
	Frm13Ctrl AT %Q* : UINT;
	{attribute addProperty Name "Frm13WcCtrl"}
	Frm13WcCtrl AT %Q* : UINT;
	{attribute addProperty Name "Frm14Ctrl"}
	Frm14Ctrl AT %Q* : UINT;
	{attribute addProperty Name "Frm14WcCtrl"}
	Frm14WcCtrl AT %Q* : UINT;
	{attribute addProperty Name "Frm15Ctrl"}
	Frm15Ctrl AT %Q* : UINT;
	{attribute addProperty Name "Frm15WcCtrl"}
	Frm15WcCtrl AT %Q* : UINT;
	{attribute addProperty Name "Frm16Ctrl"}
	Frm16Ctrl AT %Q* : UINT;
	{attribute addProperty Name "Frm16WcCtrl"}
	Frm16WcCtrl AT %Q* : UINT;
	{attribute addProperty Name "Frm17Ctrl"}
	Frm17Ctrl AT %Q* : UINT;
	{attribute addProperty Name "Frm17WcCtrl"}
	Frm17WcCtrl AT %Q* : UINT;
	{attribute addProperty Name "Frm18Ctrl"}
	Frm18Ctrl AT %Q* : UINT;
	{attribute addProperty Name "Frm18WcCtrl"}
	Frm18WcCtrl AT %Q* : UINT;
	{attribute addProperty Name "Frm19Ctrl"}
	Frm19Ctrl AT %Q* : UINT;
	{attribute addProperty Name "Frm19WcCtrl"}
	Frm19WcCtrl AT %Q* : UINT;
	{attribute addProperty Name "Frm20Ctrl"}
	Frm20Ctrl AT %Q* : UINT;
	{attribute addProperty Name "Frm20WcCtrl"}
	Frm20WcCtrl AT %Q* : UINT;
	{attribute addProperty Name "Frm21Ctrl"}
	Frm21Ctrl AT %Q* : UINT;
	{attribute addProperty Name "Frm21WcCtrl"}
	Frm21WcCtrl AT %Q* : UINT;
	{attribute addProperty Name "Frm22Ctrl"}
	Frm22Ctrl AT %Q* : UINT;
	{attribute addProperty Name "Frm22WcCtrl"}
	Frm22WcCtrl AT %Q* : UINT;
	{attribute addProperty Name "Frm23Ctrl"}
	Frm23Ctrl AT %Q* : UINT;
	{attribute addProperty Name "Frm23WcCtrl"}
	Frm23WcCtrl AT %Q* : UINT;
	{attribute addProperty Name "Frm24Ctrl"}
	Frm24Ctrl AT %Q* : UINT;
	{attribute addProperty Name "Frm24WcCtrl"}
	Frm24WcCtrl AT %Q* : UINT;
	{attribute addProperty Name "Frm25Ctrl"}
	Frm25Ctrl AT %Q* : UINT;
	{attribute addProperty Name "Frm25WcCtrl"}
	Frm25WcCtrl AT %Q* : UINT;
END_STRUCT
END_TYPE

// ---- DUTs/IO/Boxes/EK1100_1FC0878B.TcDUT
{attribute 'GeneratedUsingTerminal: EK1100-0000-0018'}
{attribute addProperty BoxType "EK1100-0000-0018"}
{attribute addProperty Description "EK1100 EtherCAT Coupler (2A E-Bus)"}
{attribute addProperty Physics "YKY"}
{attribute addProperty Id "InfoDataAT %I*InfoData_6F19DB2B2"}
{attribute addProperty CRC "532711307"}
{attribute addProperty Size "2"}
TYPE EK1100_1FC0878B EXTENDS EtcSlaveBoxBase_77A0E4A7 :
STRUCT
	{attribute addProperty Name "InfoData"}
	InfoData : InfoData_6F19DB2B;
END_STRUCT
END_TYPE

// ---- DUTs/IO/Boxes/EK1122_1FC0878B.TcDUT
{attribute 'GeneratedUsingTerminal: EK1122-0000-0018'}
{attribute addProperty BoxType "EK1122-0000-0018"}
{attribute addProperty Description "EK1122 2 port EtherCAT junction"}
{attribute addProperty Physics "KYKY"}
{attribute addProperty Id "InfoDataAT %I*InfoData_6F19DB2B2"}
{attribute addProperty CRC "532711307"}
{attribute addProperty Size "2"}
TYPE EK1122_1FC0878B EXTENDS EtcSlaveTerminalBase_947E5A46 :
STRUCT
	{attribute addProperty Name "InfoData"}
	InfoData : InfoData_6F19DB2B;
END_STRUCT
END_TYPE

// ---- DUTs/IO/Boxes/EQ1008_78E8D3DD.TcDUT
{attribute 'GeneratedUsingTerminal: EQ1008-0002-0016'}
{attribute addProperty BoxType "EQ1008-0002-0016"}
{attribute addProperty Description "EQ1008-0002 8 Ch. Dig. Input 24V, 3ms, M12"}
{attribute addProperty Physics "YY"}
{attribute addProperty Id "Channel_1AT %I*Channel_830843C11Channel_2AT %I*Channel_830843C11Channel_3AT %I*Channel_830843C11Channel_4AT %I*Channel_830843C11Channel_5AT %I*Channel_830843C11Channel_6AT %I*Channel_830843C11Channel_7AT %I*Channel_830843C11Channel_8AT %I*Channel_830843C11WcStateAT %I*WcState_9091E0EB2InfoDataAT %I*InfoData_6F19DB2B2"}
{attribute addProperty CRC "2028524509"}
{attribute addProperty Size "12"}
TYPE EQ1008_78E8D3DD EXTENDS EtcSlaveBoxBase_77A0E4A7 :
STRUCT
	{attribute addProperty Name "Channel_1"}
	Channel_1 : Channel_830843C1;
	{attribute addProperty Name "Channel_2"}
	Channel_2 : Channel_830843C1;
	{attribute addProperty Name "Channel_3"}
	Channel_3 : Channel_830843C1;
	{attribute addProperty Name "Channel_4"}
	Channel_4 : Channel_830843C1;
	{attribute addProperty Name "Channel_5"}
	Channel_5 : Channel_830843C1;
	{attribute addProperty Name "Channel_6"}
	Channel_6 : Channel_830843C1;
	{attribute addProperty Name "Channel_7"}
	Channel_7 : Channel_830843C1;
	{attribute addProperty Name "Channel_8"}
	Channel_8 : Channel_830843C1;
	{attribute addProperty Name "WcState"}
	WcState : WcState_9091E0EB;
	{attribute addProperty Name "InfoData"}
	InfoData : InfoData_6F19DB2B;
END_STRUCT
END_TYPE

// ---- DUTs/IO/Boxes/EQ1809_32157CFD.TcDUT
{attribute 'GeneratedUsingTerminal: EQ1809-0022-0016'}
{attribute addProperty BoxType "EQ1809-0022-0016"}
{attribute addProperty Description "EQ1809-0022 16 Ch. Dig. Input 24V, 3ms, M12"}
{attribute addProperty Physics "YY"}
{attribute addProperty Id "Channel_1AT %I*Channel_830843C11Channel_2AT %I*Channel_830843C11Channel_3AT %I*Channel_830843C11Channel_4AT %I*Channel_830843C11Channel_5AT %I*Channel_830843C11Channel_6AT %I*Channel_830843C11Channel_7AT %I*Channel_830843C11Channel_8AT %I*Channel_830843C11Channel_9AT %I*Channel_830843C11Channel_10AT %I*Channel_830843C11Channel_11AT %I*Channel_830843C11Channel_12AT %I*Channel_830843C11Channel_13AT %I*Channel_830843C11Channel_14AT %I*Channel_830843C11Channel_15AT %I*Channel_830843C11Channel_16AT %I*Channel_830843C11WcStateAT %I*WcState_9091E0EB2InfoDataAT %I*InfoData_6F19DB2B2"}
{attribute addProperty CRC "840269053"}
{attribute addProperty Size "20"}
TYPE EQ1809_32157CFD EXTENDS EtcSlaveBoxBase_77A0E4A7 :
STRUCT
	{attribute addProperty Name "Channel_1"}
	Channel_1 : Channel_830843C1;
	{attribute addProperty Name "Channel_2"}
	Channel_2 : Channel_830843C1;
	{attribute addProperty Name "Channel_3"}
	Channel_3 : Channel_830843C1;
	{attribute addProperty Name "Channel_4"}
	Channel_4 : Channel_830843C1;
	{attribute addProperty Name "Channel_5"}
	Channel_5 : Channel_830843C1;
	{attribute addProperty Name "Channel_6"}
	Channel_6 : Channel_830843C1;
	{attribute addProperty Name "Channel_7"}
	Channel_7 : Channel_830843C1;
	{attribute addProperty Name "Channel_8"}
	Channel_8 : Channel_830843C1;
	{attribute addProperty Name "Channel_9"}
	Channel_9 : Channel_830843C1;
	{attribute addProperty Name "Channel_10"}
	Channel_10 : Channel_830843C1;
	{attribute addProperty Name "Channel_11"}
	Channel_11 : Channel_830843C1;
	{attribute addProperty Name "Channel_12"}
	Channel_12 : Channel_830843C1;
	{attribute addProperty Name "Channel_13"}
	Channel_13 : Channel_830843C1;
	{attribute addProperty Name "Channel_14"}
	Channel_14 : Channel_830843C1;
	{attribute addProperty Name "Channel_15"}
	Channel_15 : Channel_830843C1;
	{attribute addProperty Name "Channel_16"}
	Channel_16 : Channel_830843C1;
	{attribute addProperty Name "WcState"}
	WcState : WcState_9091E0EB;
	{attribute addProperty Name "InfoData"}
	InfoData : InfoData_6F19DB2B;
END_STRUCT
END_TYPE

// ---- DUTs/IO/Boxes/EQ2008_E2806B95.TcDUT
{attribute 'GeneratedUsingTerminal: EQ2008-0002-0016'}
{attribute addProperty BoxType "EQ2008-0002-0016"}
{attribute addProperty Description "EQ2008-0002 8 Ch. Dig. Output 24V, 0,5A, M12"}
{attribute addProperty Physics "YY"}
{attribute addProperty Id "Channel_1AT %Q*Channel_42CA91F71Channel_2AT %Q*Channel_42CA91F71Channel_3AT %Q*Channel_42CA91F71Channel_4AT %Q*Channel_42CA91F71Channel_5AT %Q*Channel_42CA91F71Channel_6AT %Q*Channel_42CA91F71Channel_7AT %Q*Channel_42CA91F71Channel_8AT %Q*Channel_42CA91F71WcStateAT %I*WcState_0B2B16F91InfoDataAT %I*InfoData_6F19DB2B2"}
{attribute addProperty CRC "3800066965"}
{attribute addProperty Size "11"}
TYPE EQ2008_E2806B95 EXTENDS EtcSlaveBoxBase_77A0E4A7 :
STRUCT
	{attribute addProperty Name "Channel_1"}
	Channel_1 : Channel_42CA91F7;
	{attribute addProperty Name "Channel_2"}
	Channel_2 : Channel_42CA91F7;
	{attribute addProperty Name "Channel_3"}
	Channel_3 : Channel_42CA91F7;
	{attribute addProperty Name "Channel_4"}
	Channel_4 : Channel_42CA91F7;
	{attribute addProperty Name "Channel_5"}
	Channel_5 : Channel_42CA91F7;
	{attribute addProperty Name "Channel_6"}
	Channel_6 : Channel_42CA91F7;
	{attribute addProperty Name "Channel_7"}
	Channel_7 : Channel_42CA91F7;
	{attribute addProperty Name "Channel_8"}
	Channel_8 : Channel_42CA91F7;
	{attribute addProperty Name "WcState"}
	WcState : WcState_0B2B16F9;
	{attribute addProperty Name "InfoData"}
	InfoData : InfoData_6F19DB2B;
END_STRUCT
END_TYPE

